// TIA Portal V17 program export: 22 tag tables, 7 data types, 16 data blocks, 26 code blocks (in call order from the OBs), 29 instance data blocks

VAR_GLOBAL   // PLC tag table "Data Costant"
END_VAR
VAR_GLOBAL CONSTANT   // user constants
   MaxCreateNFP : Int := 10;   // Number of max creating NFP²s
   MaxDataReading : Int := 25;   // Number of max data reading
   MaxRoundNumber : Int := 1;   // Number of Rounds
   NumberOfmessages : Int := 6;   // Number of messages from IJCore
   MaxStageStep : Int := 25;   // Number of Max Step Step
   MaxInitStep : Int := 2;   // Number of Max Init Step
   MaxRobot : Int := 3;   // Number of Max Robot
   MaxReader : Int := 5;   // Number of Max Reader
   MaxSolenoid : Int := 48;   // Number of Max Solenoid
   NotUsed : Int := 0;
   MasterNFP : Int := 2;
   SecondaryNFP : Int := 3;
   Component : Int := 4;
   STA : Int := 1;
   PFC : Int := 2;
   TRW : Int := 3;
   TRI : Int := 4;
   TRR : Int := 5;
   CMA : Int := 7;
   TMA : Int := 8;
   CNF : Int := 9;
   TRC : Int := 10;
   TRS : Int := 6;
   TRB : Int := 11;
END_VAR

VAR_GLOBAL   // PLC tag table "Default tag table"
   optoSignal AT %I0.7 : Bool;
   nestScannerBusy AT %I3.0 : Bool;
   nestScannerComplete AT %I4.0 : Bool;
   nestScannerError AT %I5.0 : Bool;
   nestScannerDataSize AT %IW334 : Int;
   upperScannerReading AT %I9.0 : Bool;
   upperScannerReadingComplete AT %I10.0 : Bool;
   upperScannerError AT %I11.0 : Bool;
   upperScannerDataSize AT %IW470 : Int;
   angleScannerDataSize AT %IW385 : Int;
   angleScannerBusy AT %I39.0 : Bool;
   angleScannerReadingComplete AT %I40.0 : Bool;
   angleScannerError AT %I41.0 : Bool;
   amgeScannerDataSize AT %IW606 : Int;
   Tag_1 AT %I46.3 : Bool;
   Tag_2 AT %I46.4 : Bool;
   washerPresence AT %I1.0 : Bool;
   toolingID2 AT %I1.6 : Bool;
   finalTorqueAngle AT %IW17 : Word;
   OutputPin2 AT %QB147 : Byte;
   byte0 AT %QB156 : Byte;
   runlight AT %Q159.2 : Bool;
   byte6 AT %QB162 : Byte;
   byte2 AT %QB158 : Byte;
   byte7 AT %QB163 : Byte;
   segmentLight AT %Q159.0 : Bool;
   byte1 AT %QB157 : Byte;
   byte4 AT %QB160 : Byte;
   byte3 AT %QB159 : Byte;
   byte5 AT %QB161 : Byte;
   optoGreen AT %Q1.2 : Bool;
   optoRed AT %Q1.3 : Bool;
   optoYellow AT %Q1.4 : Bool;
   qYellowTurretBlinking AT %Q2.1 : Bool;
   nestScannerRequest AT %Q3.0 : Bool;
   clearUpperScannerReadComplete AT %Q9.0 : Bool;
   upperScannerRequest AT %Q8.0 : Bool;
   angleScannerRequest AT %Q13.0 : Bool;
   clearAngleScannerComplete AT %Q14.0 : Bool;
   clearTorque AT %Q17.5 : Bool;
   System_Byte AT %MB0 : Byte;
   DiagStatusUpdate AT %M0.1 : Bool;
   "CONFIG INICIAL" AT %M89.5 : Bool;
   "CONFIG CILINDROS ON" AT %M89.7 : Bool;
END_VAR
VAR_GLOBAL CONSTANT   // user constants
   "MODELO MOTOR 1" : String := '592';
   "MODELO MOTOR 2" : String := '202';
   "MODELO MOTOR 3" : String := '277';
   "MODELO MOTOR 4" : String := '984';
   "MODELO TRACK L 1" : String := '610';
   "MODELO TRACK L 2" : String := '618';
   "MODELO TRACK L 3" : String := '333';
   "MODELO TRACK L 4" : String := '444';
   "MODELO TRACK L 5" : String := '555';
   "MODELO TRACK L 6" : String := '666';
   "MODELO TRACK L 7" : String := '777';
   "MODELO TRACK L 8" : String := '888';
   "MODELO TRACK R 1" : String := '612';
   "MODELO TRACK R 2" : String := '623';
   "MODELO TRACK R 3" : String := '993';
   "MODELO TRACK R 4" : String := '994';
   "MODELO TRACK R 5" : String := '995';
   "MODELO TRACK R 6" : String := '996';
   "MODELO TRACK R 7" : String := '997';
   "MODELO TRACK R 8" : String := '998';
END_VAR

VAR_GLOBAL   // PLC tag table "EKSMemory"
   eksUserLevel AT %MB2101 : SInt;
   ActualAuthorizationLevel AT %MB2100 : SInt;
   electronicKeyPresent AT %MB2102 : SInt;
END_VAR

VAR_GLOBAL   // PLC tag table "alarmMemory"
   alarm0 AT %MW100 : Int;   // alarm number
   alarm1 AT %MW102 : Int;   // alarm number
   alarm2 AT %MW104 : Int;
   retIolink AT %MW108 : Int;
   retManifold AT %MW112 : Int;
   retEuchner AT %MW106 : Int;
   retIolink2 AT %MW110 : Int;
   removeScannerError AT %MW6 : Word;
   Green AT %M2.0 : Bool;
   yellow AT %M2.1 : Bool;
   red AT %M2.2 : Bool;
   qRedTurretSolid AT %M3.6 : Bool;
   kkkk AT %M8.1 : Bool;
   hmifinalTorqueAngle AT %MW10 : Word;
END_VAR

VAR_GLOBAL   // PLC tag table "clockMemory"
   Clock_Byte AT %MB1 : Byte;
   Clocks_100ms_FP AT %M1.0 : Bool;
   Clocks_200ms_FP AT %M1.1 : Bool;
   Clocks_400ms_FP AT %M1.2 : Bool;
   Clocks_500ms_FP AT %M1.3 : Bool;
   Clocks_800ms_FP AT %M1.4 : Bool;
   Clocks_1s_FP AT %M1.5 : Bool;
   Clocks_1S600ms_FP AT %M1.6 : Bool;
   Clocks_2s_FP AT %M1.7 : Bool;
END_VAR

VAR_GLOBAL   // PLC tag table "codeReaderMemory"
   reqScannerConfig AT %M2250.2 : Bool;
   bufferReset AT %M2250.0 : Bool;
   labelReadingError AT %M186.3 : Bool;
   labelNok AT %M187.0 : Bool;
   nestLabelReadingError AT %M224.0 : Bool;
   idleTime AT %M2250.1 : Bool;
   seatLabelIdentified AT %M2250.3 : Bool;
   motorLabelIdentified AT %M2250.4 : Bool;
   xLabelIdentified AT %M2250.5 : Bool;
   hmiNestScannerReq AT %M2.3 : Bool;
   scannerOnConfig AT %M2.6 : Bool;
   scanningNest AT %M2.7 : Bool;
   nestCodeRead AT %M3.3 : Bool;
   upperScannerCodeRead AT %M3.4 : Bool;
   angleScannerCodeRead AT %M3.7 : Bool;
   scanningAngle AT %M4.2 : Bool;
   scanningUpper AT %M4.6 : Bool;
   label1Upper AT %M8.2 : Bool;
   label2Upper AT %M8.3 : Bool;
END_VAR

VAR_GLOBAL   // PLC tag table "hmiMemory"
   currentModel AT %MW3000 : Int;
   hmiButtonVisualization AT %M3050.6 : Bool;
   previousModel AT %MW3008 : Int;
   currentStep AT %MW3002 : Int;
   numbersOfStepsToMove AT %MW3006 : UInt;
   stepToDivide AT %MW3012 : UInt;
   stepToInsert AT %MW3014 : UInt;
   hmiScreenNumber AT %MW22 : Int;
   allowedTextChange AT %M3050.0 : Bool;
   progressBarMultiply AT %MW3010 : Int;
   lastCycleInputs AT %MD3034 : DInt;
   energySavingElapsedTime AT %MD3030 : Time;
   f7Button AT %M3050.5 : Bool;
   sequencerCopySequence AT %M66.2 : Bool;
   codeReaderConfigurationVisible AT %M3050.2 : Bool;
   directAlarm AT %M3050.3 : Bool;
   directHome AT %M3050.4 : Bool;
   saveHMI AT %M2.4 : Bool;
   readHMI AT %M2.5 : Bool;
   home AT %M4.7 : Bool;
   ready4Movement AT %M5.5 : Bool;
   popUpVisible AT %M5.6 : Bool;
END_VAR

VAR_GLOBAL   // PLC tag table "modeMemory"
   automaticMode AT %M3.0 : Bool;   // AUTO = 1
   manualMode AT %M3.1 : Bool;
   noMode AT %M3.2 : Bool;
   modelChangePermit AT %M187.1 : Bool;
END_VAR

VAR_GLOBAL   // PLC tag table "permissionMemory"
   MaintenacePermission AT %M4.4 : Bool;
   adminPermission AT %M4.0 : Bool;
   lgPermission AT %M4.5 : Bool;
   gapLeaderUser AT %M4.3 : Bool;
   editingPermission AT %M4.1 : Bool;
   confirmStandby AT %M5.7 : Bool;
   cancelMovement AT %M8.0 : Bool;
END_VAR

VAR_GLOBAL   // PLC tag table "productionMemory"
   shift1Production AT %MW300 : Int;
   shift1 AT %M350.0 : Bool;
   shift2Production AT %MW302 : Int;
   shift2 AT %M350.1 : Bool;
   shift3Production AT %MW304 : Int;
   shift3 AT %M350.2 : Bool;
   timeShift1 AT %M350.3 : Bool;
   timeShift2 AT %M350.4 : Bool;
   timeShift3 AT %M350.5 : Bool;
END_VAR

VAR_GLOBAL   // PLC tag table "programMemory"
   cycleTimeReset AT %M250.1 : Bool;
   clearData AT %M250.0 : Bool;
   productInNest AT %M250.2 : Bool;
   programAutoModeSelection AT %M250.3 : Bool;
END_VAR

VAR_GLOBAL   // PLC tag table "pulses"
   startTighteningPulse1 AT %Q124.0 : Bool;
   hmiPulseInt AT %MD2000 : DInt;
   hmiCycleCounterRestartPulse AT %M2004.4 : Bool;
   model01SelectedPulse AT %M2004.6 : Bool;
   model02SelectedPulse AT %M2004.7 : Bool;
   model03SelectedPulse AT %M2005.0 : Bool;
   model04SelectedPulse AT %M2005.1 : Bool;
   model05SelectedPulse AT %M2005.2 : Bool;
   model06SelectedPulse AT %M2005.3 : Bool;
   model07SelectedPulse AT %M2005.4 : Bool;
   model08SelectedPulse AT %M2005.5 : Bool;
   model09SelectedPulse AT %M2005.6 : Bool;
   model10SelectedPulse AT %M2005.7 : Bool;
   model11SelectedPulse AT %M2006.0 : Bool;
   model12SelectedPulse AT %M2006.1 : Bool;
   mode13SelectedPulse AT %M2006.2 : Bool;
   mode14SelectedPulse AT %M2006.3 : Bool;
   mode15SelectedPulse AT %M2006.4 : Bool;
   alarmPresPulse AT %M2004.3 : Bool;
   "1stShiftChangePulse" AT %M2004.0 : Bool;
   "2ndShiftChangePulse" AT %M2004.1 : Bool;
   "3rdShiftChangePulse" AT %M2004.2 : Bool;
   stepChangeTimerResetInputPulse AT %M2009.4 : Bool;
   stepChangeTimerResetOutputPulse AT %M2009.5 : Bool;
   stationTurnedOffInSequencePulse AT %M2009.3 : Bool;
   model32SelectedPulse AT %M2008.5 : Bool;
   model31SelectedPulse AT %M2008.4 : Bool;
   model30SelectedPulse AT %M2008.3 : Bool;
   model29SelectedPulse AT %M2008.2 : Bool;
   model27SelectedPulse AT %M2008.0 : Bool;
   model28SelectedPulse AT %M2008.1 : Bool;
   model26SelectedPulse AT %M2007.7 : Bool;
   model25SelectedPulse AT %M2007.6 : Bool;
   model24SelectedPulse AT %M2007.5 : Bool;
   model23SelectedPulse AT %M2007.4 : Bool;
   model22SelectedPulse AT %M2007.3 : Bool;
   model21SelectedPulse AT %M2007.2 : Bool;
   model20SelectedPulse AT %M2007.1 : Bool;
   model19SelectedPulse AT %M2007.0 : Bool;
   model18SelectedPulse AT %M2006.7 : Bool;
   model17SelectedPulse AT %M2006.6 : Bool;
   model16SelectedPulse AT %M2006.5 : Bool;
   scanner3DataLogPulse AT %M2009.2 : Bool;
   scanner2DataLogPulse AT %M2009.1 : Bool;
   scanner1DataLogPulse AT %M2009.0 : Bool;
   rightTrackScannerPulse AT %M2008.7 : Bool;
   leftTrackScannerPulse AT %M2004.5 : Bool;
   motorScannerPulse AT %M2008.6 : Bool;
   clearDataPulse AT %M2010.0 : Bool;
   hmiCylinderPulse AT %M5.4 : Bool;
END_VAR

VAR_GLOBAL   // PLC tag table "sequenceMemory"
   aa AT %MW24 : Int;
   a_correctas AT %MW32 : Int;
   a_estados AT %MW34 : Int;
   verificacion_estados_A AT %MW44 : Int;
   verificacion_estados_B AT %MW26 : Int;
   b_estados AT %MW36 : Int;
   numberOfCorrectOutputStates AT %MW38 : Int;
   bb AT %MW40 : Int;
   previousStep AT %MW1112 : Int;
   sequenceRestart AT %M89.1 : Bool;
   stationTurnedOffInSequence AT %M1150.1 : Bool;
END_VAR

VAR_GLOBAL   // PLC tag table "systemMemory"
   firstScan AT %M0.0 : Bool;
   LOG0 AT %M0.3 : Bool;
   LOG1 AT %M0.2 : Bool;
END_VAR

VAR_GLOBAL   // PLC tag table "EKSFieldbusInputs"
   iEKSLevel AT %IB201 : Byte;
   iEKSChipInside AT %I200.1 : Bool;
   iEKSEmpolyeeNumber AT %ID221 : DWord;
   iEKSKeyID1 AT %ID320 : DWord;
   iEKSKeyID2 AT %ID324 : DWord;
   iEKSEmployeeNumber AT %I200.6 : Bool;
   usserIsLogged AT %M2150.0 : Bool;
END_VAR

VAR_GLOBAL   // PLC tag table "powerFocus6000"
   counterClockwiseDirection AT %I182.5 : Bool;
   clockwiseDirection AT %I182.6 : Bool;
   torqueOk AT %I19.6 : Bool;
   torqueDone AT %I20.0 : Bool;
   torqueNok AT %I19.7 : Bool;
   finalTorqueInt1 AT %IW13 : Word;
   finalTorqueDecimal1 AT %IW15 : Word;
   deactivateTool AT %Q17.7 : Bool;
   activateTorqueTool AT %Q17.0 : Bool;
   clearNestScanerRead AT %Q4.0 : Bool;
   torqueInputSelect AT %QB18 : Byte;
   thighteningStart AT %Q17.3 : Bool;
   correctTorque AT %M3.5 : Bool;
   p6000Test1 AT %M152.1 : Bool;
   p6000Test2 AT %M152.2 : Bool;
   p6000Test3 AT %M152.3 : Bool;
   p6000Test1Enabled AT %M152.4 : Bool;
   p6000Test2Enabled AT %M152.5 : Bool;
   p6000Test3Enabled AT %M152.6 : Bool;
   counterClockwiseDirectionWarning AT %M23.0 : Bool;
   clockwiseDirectionWarning AT %M23.1 : Bool;
   hmiFinalTorqueDecimal AT %MW214 : Word;
   hmiFinalTorqueInt AT %MW212 : Word;
END_VAR

VAR_GLOBAL   // PLC tag table "safetyControllerFieldbusInputs"
   isecurityEnabled AT %I46.0 : Bool;
   iEmergencyStop AT %I46.1 : Bool;
   emergencyStopMonitor AT %I46.2 : Bool;
END_VAR

VAR_GLOBAL   // PLC tag table "digitalFieldbusInputs"
   iRightManualRodInsExt AT %I156.5 : Bool;
   iLeftToolingLockExt AT %I1.3 : Bool;
   iRightToolingExt AT %I156.7 : Bool;
   iTorqueToolingExt AT %I156.6 : Bool;
   iRigthManualRodInsRet AT %I157.5 : Bool;
   iLeftToolingLockRet AT %I1.4 : Bool;
   iRightToolingRet AT %I157.7 : Bool;
   iTorqueToolingRet AT %I157.6 : Bool;
   iStrapDetection AT %I45.3 : Bool;
   iLeftBracketDetection AT %I45.2 : Bool;
   iPresLeftManFrame AT %I157.1 : Bool;
   iRightBracketDetection AT %I45.0 : Bool;
   iManualExtOk AT %I158.3 : Bool;
   iProductInsertedLh AT %I45.1 : Bool;
   iLeftHomePos AT %I159.6 : Bool;
   iLeftWorkPos AT %I158.6 : Bool;
   iLeftToolingPos3 AT %I158.7 : Bool;
   iManualExtNok AT %I159.3 : Bool;
   iPresRightPwrFrame AT %I156.3 : Bool;
   iManualBumper AT %I158.5 : Bool;
   iLeftSpringColor AT %I158.2 : Bool;
   iRightSpringColor AT %I158.4 : Bool;
   iLeftManualRodInsRet AT %I157.4 : Bool;
   iInsertionCylindersRet AT %I1.2 : Bool;
   iInsertionCylindersExt AT %I1.1 : Bool;
   iLeftManToolingExtNok AT %I159.7 : Bool;
   iProductInsertedRh AT %I45.6 : Bool;
   iTorqueToolingHome AT %I45.5 : Bool;
   iRightToolinPos1 AT %I156.4 : Bool;
   iRightToolinPos3 AT %I156.2 : Bool;
   iRightToolinPos2 AT %I157.2 : Bool;
   iManualZExtOk AT %I156.0 : Bool;
   iManualZExtNok AT %I157.0 : Bool;
   iRightManToolingRet AT %I158.1 : Bool;
   iTorqueTrigger AT %I160.0 : Bool;
   toolingID1 AT %I1.5 : Bool;
   manualProductPres AT %Q10.0 : Bool;
   powerProductPres AT %Q10.1 : Bool;
END_VAR

VAR_GLOBAL   // PLC tag table "digitalPLCInputs"
   iAirPreassureSensor AT %I0.1 : Bool;
   iPresRightManFrame AT %I156.1 : Bool;
   iRestartButton AT %I0.0 : Bool;
END_VAR

VAR_GLOBAL   // PLC tag table "digitalFieldbusOutputs"
   qcylinder1DirectionA AT %Q149.0 : Bool;
   qcylinder1DirectionB AT %Q151.0 : Bool;
   qcylinder2DirectionA AT %Q149.1 : Bool;
   qcylinder2DirectionB AT %Q151.1 : Bool;
   qcylinder7DirectionA AT %Q701.2 : Bool;
   qcylinder7DirectionB AT %Q701.3 : Bool;
   qcylinder4DirectionA AT %Q149.3 : Bool;
   qcylinder4DirectionB AT %Q151.3 : Bool;
   qcylinder5DirectionA AT %Q149.4 : Bool;
   qcylinder5DirectionB AT %Q151.4 : Bool;
   qcylinder6DirectionA AT %Q149.5 : Bool;
   qcylinder6DirectionB AT %Q151.5 : Bool;
   qcylinder3DirectionA AT %Q149.2 : Bool;
   qcylinder3DirectionB AT %Q151.2 : Bool;
   qcylinder8DirectionA AT %Q701.4 : Bool;
   qcylinder8DirectionB AT %Q701.5 : Bool;
   qcylinder9DirectionA AT %Q701.6 : Bool;
   qcylinder9DirectionB AT %Q701.7 : Bool;
   qcylinder10DirectionA AT %Q702.0 : Bool;
   qcylinder10DirectionB AT %Q702.1 : Bool;
   qActivateCutOffValve AT %Q147.7 : Bool;
END_VAR

VAR_GLOBAL   // PLC tag table "digitalPLCOutputs"
   qAirInletValve1 AT %Q0.0 : Bool;
   qLampActivation AT %Q1.0 : Bool;
   qFanActivation AT %Q1.1 : Bool;
   qControlIN AT %Q1.7 : Bool;
   qAirInletValve2 AT %Q0.1 : Bool;
   qRedTurretBlinking AT %M5.0 : Bool;
   qYellowTurretSolid AT %M5.1 : Bool;
   qGreenTurret AT %M5.2 : Bool;
   qBlueTurret AT %M5.3 : Bool;
END_VAR

VAR_GLOBAL   // PLC tag table "EKSFieldbusOutputs"
   qEKSStartAddress AT %QB201 : Byte;
   qEKSDataLength AT %QB202 : Byte;
   qEKSData1 AT %QB204 : Byte;
   qEKSData2 AT %QB205 : Byte;
   qEKsWriteCMD AT %Q200.0 : Bool;
END_VAR

TYPE "UDT_Readings"
// stored: IsFailsafeCompliant false
   STRUCT
      Enable : Bool;   // Reading active
      ReaderNumber : USInt;   // Fix (1 to 5) or Manual (10)
      "Name" : String[30];   // Name of Label to read
      LabelType : USInt;   // Master NFP, 2nd NFP, Component Label, batch label
      ReferenceToFound : String[30];   // Reference to be found
      ReferenceStartPosition : USInt;   // Position of reference to be found
      ReferenceLenght : USInt;   // Reference Lenght
      MasterReadingNumber : USInt;   // Reading number of master NFP
      LinkedMasterNumber : USInt;   // Linked number to master NFP
      Message : Array[1.."NumberOfmessages"] of "UDT_IJCoreMessage";   // IJCore Message
   END_STRUCT;
END_TYPE

TYPE "UDT_ScrewData"
// stored: IsFailsafeCompliant false
   STRUCT
      Torque : Struct   // Torque Data
         BeforePoint : Word;   // Torque before point
         AfterPoint : Word;   // Torque after point
      END_STRUCT;
      Angle : Word;   // angle
   END_STRUCT;
END_TYPE

TYPE "udtButtons"
// stored: IsFailsafeCompliant false
   STRUCT
      bReq : Bool;
      bP : Bool;
      bTGG : Bool;
      bCmd : Bool;
      bAkn : Bool;
      b1 : Bool;
      b2 : Bool;
      b3 : Bool;
   END_STRUCT;
END_TYPE

TYPE "udt_EKS_KEY"
// stored: IsFailsafeCompliant false
   STRUCT
      ID1 : DWord;   // Key unique ID [bytes 1-4]
      ID2 : DWord;   // Key unique ID [bytes 5-8]
      EMPLOYEE_ID : DWord;   // Employee ID number [hex format]
      LEVEL : Int;   // Key level stored inside key
      COMMENTS : WString[10];   // Comments of the key
      _res_1 : Int;
   END_STRUCT;
END_TYPE

TYPE "udt_referenceMainInfo"
// stored: IsFailsafeCompliant false
   STRUCT
      id : Int;
      description : String[20];
      partNumber : String[8];
      rev : String[2];
      customerNumber : String[8];
      vpps : String[14];
      locationCode : String[1];
      dataIdentifier : String[3];
      duns : String[9];
   END_STRUCT;
END_TYPE

TYPE "CONFIG_MSG_IJC"
// stored: IsFailsafeCompliant false
   STRUCT
      "TYPE" : String[3];
      KANBAN : String[30];
      COMPONENT : String[62];
      START : Bool;
      PROCESS_STATUS : SInt;
   END_STRUCT;
END_TYPE

TYPE "UDT_IJCoreMessage"
// stored: IsFailsafeCompliant false
   STRUCT
      MessageType : USInt;
      MessageFlagNumber : UInt;
      SendMsg : Bool;
      Done : Bool;
      Answer : Int;
      State : USInt;
   END_STRUCT;
END_TYPE

DATA_BLOCK "DB_MAIN_IJCORE"   // DB1000
{ S7_Optimized_Access := 'FALSE' }
VERSION : 0.1
// stored: AutoNumber false, DBAccessibleFromOPCUA true, DBAccessibleFromWebserver true, IsOnlyStoredInLoadMemory false, IsWriteProtectedInAS false
   VAR
      Enable : Bool := true;   // Enable traceability
      Mode : USInt := 1;   // 1. Full traceability, 2. Downgrade Mode
      Errors : Word;   // Error code
      hmiInd : USInt;   // Global Indicator Status
      CreatedNFP : Array[1.."MaxCreateNFP"] of String[30];   // Created NFP
      STAT : Struct
         STA_OK : Bool;
         PFC_OK : Bool;
         TRC_OK : Bool;
         CNF_OK : Bool;
         TRR_OK : Bool;
         ProcessResults : USInt;   // 1: Part OK, 2: PartNOK
      END_STRUCT;
      CMD : Struct
         STA : Bool;
         PFC : Bool;
         TRC : Bool;
         CNF : Bool;
         TRR : Bool;
      END_STRUCT;
   END_VAR
BEGIN
END_DATA_BLOCK

DATA_BLOCK "DB_REC_IJCORE"   // DB1006
{ S7_Optimized_Access := 'FALSE' }
VERSION : 0.1
// stored: AutoNumber false, DBAccessibleFromOPCUA true, DBAccessibleFromWebserver true, IsOnlyStoredInLoadMemory false, IsWriteProtectedInAS false
   VAR
      SW_Message : Array[1..300] of Word;
      Message : Array[1..50] of Struct
         Answer : Int;
         Content : Array[1..30] of Byte;
      END_STRUCT;
   END_VAR
BEGIN
END_DATA_BLOCK

DATA_BLOCK "DB_SEND_IJCORE"   // DB1005
{ S7_Optimized_Access := 'FALSE' }
VERSION : 0.1
// stored: AutoNumber false, DBAccessibleFromOPCUA true, DBAccessibleFromWebserver true, IsOnlyStoredInLoadMemory false, IsWriteProtectedInAS false
   VAR
      Awake_DW : Word;
      Awake_SW : Int;
      SW_Message : Array[1..300] of Word;
      Message : Array[1..50] of Struct
         Content : Array[1..80] of Byte;
      END_STRUCT;
   END_VAR
BEGIN
END_DATA_BLOCK

DATA_BLOCK "DB_EKS"   // DB305
{ S7_Optimized_Access := 'FALSE' }
VERSION : 0.1
// stored: AutoNumber false, DBAccessibleFromOPCUA true, DBAccessibleFromWebserver true, IsOnlyStoredInLoadMemory false, IsWriteProtectedInAS false
   VAR RETAIN
      STAT : Struct
         OPERATOR : Bool := TRUE;
         GAP_LEADER : Bool := TRUE;
         MAINTENANCE : Bool := TRUE;
         ADMINISTRATOR : Bool := TRUE;
         _4 : Bool := FALSE;
         _5 : Bool := FALSE;
         _6 : Bool := FALSE;
         _7 : Bool := FALSE;
         ADD_MODE_ENABLED : Bool := TRUE;
         ADD_MODE : Bool := FALSE;
         RESET : Bool := FALSE;
         NB_MAX_ACHIEVED : Bool := FALSE;
         FP_STORE_KEY_IN : Bool := FALSE;
         _15 : Bool := FALSE;
         _16 : Bool := FALSE;
         _17 : Bool := FALSE;
      END_STRUCT;
      HMI : Struct
         OPERATOR_KEY : Bool := FALSE;
         ADD_MODE : Bool := FALSE;
         END_ADD_MODE : Bool := FALSE;
         WRITE_NEW_KEY_LEVEL : Bool := FALSE;
         WRITE_NEW_KEY_ID : Bool := FALSE;
         UPDATE_NB_ADMIN : Bool := FALSE;
         _6 : Bool := FALSE;
         _7 : Bool := FALSE;
         _10 : Bool := FALSE;
         _11 : Bool := FALSE;
         _12 : Bool := FALSE;
         _13 : Bool := FALSE;
         _14 : Bool := FALSE;
         _15 : Bool := FALSE;
         _16 : Bool := FALSE;
         _17 : Bool := FALSE;
      END_STRUCT;
      TIM : Struct
         RESET_SET : Int := 9999;
         RESET_STAT : Int := 2960;
      END_STRUCT;
      PAGE_INDEX : Int := 1;   // Index of the page of HMI
      SAVE_LINE : Int := 0;   // Line to save key
      REMOVE_LINE : Int := 0;   // Line to remove key
      ACTUAL_LEVEL : Int := 5;   // Actual level of key
      NB_ADMIN : Int := 27414;   // Number of admin counted
      T_CYCLE : Int := 0;   // Index for function Cycle (look for key)
      NB_MAX_ADMIN : Int := 5;   // Number of administrator max
      Number_page_saved : Word := 16#0001;
      _res : Array[22..47] of Byte;   // Reserve
      INSERTED_KEY { S7_SetPoint := 'True'} : "udt_EKS_KEY";   // Information of Key Inserted
      HMI_PAGE { S7_SetPoint := 'True'} : Array[1..10] of "udt_EKS_KEY";   // Information displayed on HMI
      _res_1 : Array[270..299] of Byte;   // Reserve
      KEYS { S7_SetPoint := 'True'} : Array[1..130] of "udt_EKS_KEY";
      DELETE_KEY : "udt_EKS_KEY";
   END_VAR
BEGIN
   _res[22..47] := 16#00;
   INSERTED_KEY.ID1 := 16#383E_0010;
   INSERTED_KEY.ID2 := 16#3200_0000;
   INSERTED_KEY.EMPLOYEE_ID := 16#0000_0000;
   INSERTED_KEY.LEVEL := 5;
   INSERTED_KEY.COMMENTS := WSTRING#'LIMON';
   INSERTED_KEY._res_1 := 0;
   HMI_PAGE[1].ID1 := 16#2B2F_0010;
   HMI_PAGE[2].ID1 := 16#28A5_0010;
   HMI_PAGE[3].ID1 := 16#0000_0000;
   HMI_PAGE[4].ID1 := 16#71A6_0010;
   HMI_PAGE[5].ID1 := 16#8037_0010;
   HMI_PAGE[6].ID1 := 16#383E_0010;
   HMI_PAGE[7].ID1 := 16#5A1E_0010;
   HMI_PAGE[8].ID1 := 16#D65A_0010;
   HMI_PAGE[9..10].ID1 := 16#0000_0000;
   HMI_PAGE[1..2].ID2 := 16#3200_0000;
   HMI_PAGE[3].ID2 := 16#0000_0000;
   HMI_PAGE[4..8].ID2 := 16#3200_0000;
   HMI_PAGE[9..10].ID2 := 16#0000_0000;
   HMI_PAGE[1..7].EMPLOYEE_ID := 16#0000_0000;
   HMI_PAGE[8].EMPLOYEE_ID := 16#0000_0001;
   HMI_PAGE[9..10].EMPLOYEE_ID := 16#0000_0000;
   HMI_PAGE[1].LEVEL := 5;
   HMI_PAGE[2].LEVEL := 3;
   HMI_PAGE[3].LEVEL := 0;
   HMI_PAGE[4].LEVEL := 2;
   HMI_PAGE[5].LEVEL := 3;
   HMI_PAGE[6].LEVEL := 5;
   HMI_PAGE[7].LEVEL := 3;
   HMI_PAGE[8].LEVEL := 2;
   HMI_PAGE[9..10].LEVEL := 0;
   HMI_PAGE[1].COMMENTS := WSTRING#'CLAUDIO';
   HMI_PAGE[2].COMMENTS := WSTRING#'CLAUDIO-M';
   HMI_PAGE[3].COMMENTS := WSTRING#'';
   HMI_PAGE[4].COMMENTS := WSTRING#'GAP-1';
   HMI_PAGE[5].COMMENTS := WSTRING#'MANT-1';
   HMI_PAGE[6].COMMENTS := WSTRING#'LIMON';
   HMI_PAGE[7].COMMENTS := WSTRING#'MANT';
   HMI_PAGE[8].COMMENTS := WSTRING#'GAP';
   HMI_PAGE[9..10].COMMENTS := WSTRING#'';
   HMI_PAGE[1..10]._res_1 := 0;
   _res_1[270..299] := 16#00;
   KEYS[1].ID1 := 16#2B2F_0010;
   KEYS[2].ID1 := 16#28A5_0010;
   KEYS[3].ID1 := 16#0000_0000;
   KEYS[4].ID1 := 16#71A6_0010;
   KEYS[5].ID1 := 16#8037_0010;
   KEYS[6].ID1 := 16#383E_0010;
   KEYS[7].ID1 := 16#5A1E_0010;
   KEYS[8].ID1 := 16#D65A_0010;
   KEYS[9..109].ID1 := 16#0000_0000;
   KEYS[110].ID1 := 16#DB52_0010;
   KEYS[111..130].ID1 := 16#0000_0000;
   KEYS[1..2].ID2 := 16#3200_0000;
   KEYS[3].ID2 := 16#0000_0000;
   KEYS[4..8].ID2 := 16#3200_0000;
   KEYS[9..109].ID2 := 16#0000_0000;
   KEYS[110].ID2 := 16#3200_0000;
   KEYS[111..130].ID2 := 16#0000_0000;
   KEYS[1..7].EMPLOYEE_ID := 16#0000_0000;
   KEYS[8].EMPLOYEE_ID := 16#0000_0001;
   KEYS[9..130].EMPLOYEE_ID := 16#0000_0000;
   KEYS[1].LEVEL := 5;
   KEYS[2].LEVEL := 3;
   KEYS[3].LEVEL := 0;
   KEYS[4].LEVEL := 2;
   KEYS[5].LEVEL := 3;
   KEYS[6].LEVEL := 5;
   KEYS[7].LEVEL := 3;
   KEYS[8].LEVEL := 2;
   KEYS[9..109].LEVEL := 0;
   KEYS[110].LEVEL := 5;
   KEYS[111..130].LEVEL := 0;
   KEYS[1].COMMENTS := WSTRING#'CLAUDIO';
   KEYS[2].COMMENTS := WSTRING#'CLAUDIO-M';
   KEYS[3].COMMENTS := WSTRING#'';
   KEYS[4].COMMENTS := WSTRING#'GAP-1';
   KEYS[5].COMMENTS := WSTRING#'MANT-1';
   KEYS[6].COMMENTS := WSTRING#'LIMON';
   KEYS[7].COMMENTS := WSTRING#'MANT';
   KEYS[8].COMMENTS := WSTRING#'GAP';
   KEYS[9..109].COMMENTS := WSTRING#'';
   KEYS[110].COMMENTS := WSTRING#'Robins';
   KEYS[111..130].COMMENTS := WSTRING#'';
   KEYS[1..130]._res_1 := 0;
   DELETE_KEY.ID1 := 16#0000_0000;
   DELETE_KEY.ID2 := 16#0000_0000;
   DELETE_KEY.EMPLOYEE_ID := 16#0000_0000;
   DELETE_KEY.LEVEL := 0;
   DELETE_KEY.COMMENTS := WSTRING#'';
   DELETE_KEY._res_1 := 0;
END_DATA_BLOCK

DATA_BLOCK "LABELS"   // DB6
{ S7_Optimized_Access := 'TRUE' }
VERSION : 0.1
// stored: AutoNumber false, DBAccessibleFromOPCUA true, DBAccessibleFromWebserver true, IsOnlyStoredInLoadMemory false, IsRetainMemResEnabled false, IsWriteProtectedInAS false, MemoryReserve 100
   VAR
      "Previous code" : String := '[) 06 Y40.02.07.01.L P8127005 12V812785841 T9T22202A2B4C1004';
      "Result comp 3" : Int := 0;
      "Result comp 2" : Int := 0;
      "Result comp 1" : Int := 0;
      "Label comp 3" : String := '';
      "Label comp 2" : String := '';
      "Label comp 1" : String := '15';
   END_VAR
   VAR RETAIN
      "Label 1" : Array[0..16] of String[5];   // Label 1
      "Label 2" { ExternalVisible := 'False'} : Array[0..16] of String[5];
      "Label 3" : Array[0..16] of String[5];
      "Label 4" : Array[0..16] of String[5];
      "Label 5" : Array[0..16] of String[5];
      "Label Pos 1" : Array[0..16] of Int;   // label position 1
      "Label Pos 2" : Array[0..16] of Int;
      "Label Pos 3" : Array[0..16] of Int;
      "Label Pos 4" : Array[0..16] of Int;
      "Label Pos 5" : Array[0..16] of Int;   // label position 2
      "Label int" : Array[0..16] of Int;
      Text : Array[0..16] of String[10];   // label text hmi
   END_VAR
   VAR
      Done : Bool := FALSE;
      "Port error" : Bool := FALSE;
      "Port status" : Word := 16#7000;
      "Reset status" : Word := 16#7000;
   END_VAR
   VAR RETAIN
      "Reset done" : Bool := FALSE;
      scanner1 : Bool := TRUE;
      scanner2 : Bool := TRUE;
      scanner3 : Bool := TRUE;
      scanner4 : Bool := FALSE;
      scanner5 : Bool := FALSE;
      scanner6 : Bool := FALSE;
   END_VAR
   VAR
      scannerOn : Bool := TRUE;
      "scann code" : Array[0..1] of String[30];
      "Recive code 2" : String[80] := '';
      labelPrint : String[20] := 'CR24032821X05357';
      NFP : String[35] := '';
      "Recive code" : String[80] := '';
      NDR : Bool := FALSE;
      Error : Bool := FALSE;
      Status : Word := 16#7002;
      Length : UInt := 0;
      labelBlock : Array[0..6] of Bool;
      "Reading scann 1" : String[180] := '';
      "Reading scann 2" : String[180] := 'V008345Y4259698XR011464240801';
      "Extract 5" : Array[0..16] of String[10];
      "Extract 4" : Array[0..16] of String[10];
      "Extract 3" : Array[0..16] of String[10];
      "Extract 2" : Array[0..16] of String[10];
      "Extract 1" : Array[0..16] of String[10];
      "Scanner reading" : Array[0..254] of Char;
      "Previous code scann" : String[40] := '';
      scannerOK2 : Bool := FALSE;
      scannerOK3 : Bool := FALSE;
      scannerOK4 : Bool := FALSE;
      scannerOK5 : Bool := FALSE;
      ScannerOK1 : Bool := FALSE;
      "Scanner length 5" : Array[0..16] of Int;
      "Scanner length 4" : Array[0..16] of Int;
      "Scanner length 3" : Array[0..16] of Int;
      "Scanner length 2" : Array[0..16] of Int;
      "Scanner length 1" : Array[0..16] of Int;
      nestCodeRead : String[80] := '';
      upperCodeRead : String[80] := '';
      angleCodeRead : String[80] := '';
   END_VAR
BEGIN
   "Label 1"[0] := '695';
   "Label 1"[1] := '698';
   "Label 1"[2] := '695';
   "Label 1"[3] := '721';
   "Label 1"[4] := '8721X';
   "Label 1"[5..6] := '698';
   "Label 1"[7..16] := '';
   "Label 2"[0..3] := '06';
   "Label 2"[4] := '1';
   "Label 2"[5] := '06';
   "Label 2"[6] := 'Y4';
   "Label 2"[7..16] := '';
   "Label 3"[0..3] := '06';
   "Label 3"[4] := '';
   "Label 3"[5] := '06';
   "Label 3"[6..16] := '';
   "Label 4"[0..3] := 'Y4';
   "Label 4"[4] := '5/';
   "Label 4"[5] := 'Y4';
   "Label 4"[6] := '5/';
   "Label 4"[7..16] := '';
   "Label 5"[0..6] := '5/';
   "Label 5"[7..16] := '';
   "Label Pos 1"[0..3] := 13;
   "Label Pos 1"[4] := 12;
   "Label Pos 1"[5..6] := 13;
   "Label Pos 1"[7..16] := 0;
   "Label Pos 2"[0..3] := 4;
   "Label Pos 2"[4] := 1;
   "Label Pos 2"[5] := 4;
   "Label Pos 2"[6] := 1;
   "Label Pos 2"[7..16] := 0;
   "Label Pos 3"[0..3] := 4;
   "Label Pos 3"[4] := 0;
   "Label Pos 3"[5] := 4;
   "Label Pos 3"[6..16] := 0;
   "Label Pos 4"[0..3] := 1;
   "Label Pos 4"[4] := 20;
   "Label Pos 4"[5] := 1;
   "Label Pos 4"[6] := 20;
   "Label Pos 4"[7..16] := 0;
   "Label Pos 5"[0..6] := 20;
   "Label Pos 5"[7..16] := 0;
   "Label int"[0] := 151;
   "Label int"[1..16] := 0;
   Text[0] := '';
   Text[1] := 'NEST';
   Text[2] := 'UPPER1';
   Text[3] := 'ANGLE';
   Text[4] := 'UPPER2';
   Text[5..16] := '';
   "scann code"[0..1] := '';
   labelBlock[0..6] := FALSE;
   "Extract 5"[0..16] := '';
   "Extract 4"[0..16] := '';
   "Extract 3"[0..16] := '';
   "Extract 2"[0..16] := '';
   "Extract 1"[0..16] := '';
   "Scanner reading"[0] := '$L';
   "Scanner reading"[1] := '†';
   "Scanner reading"[2] := '$L';
   "Scanner reading"[3] := '†';
   "Scanner reading"[4] := '$L';
   "Scanner reading"[5] := '†';
   "Scanner reading"[6] := '$00';
   "Scanner reading"[7] := '$1E';
   "Scanner reading"[8] := 'B';
   "Scanner reading"[9..10] := '0';
   "Scanner reading"[11] := '2';
   "Scanner reading"[12] := '3';
   "Scanner reading"[13] := '9';
   "Scanner reading"[14] := '0';
   "Scanner reading"[15] := 'W';
   "Scanner reading"[16] := '4';
   "Scanner reading"[17] := '2';
   "Scanner reading"[18] := '6';
   "Scanner reading"[19] := '8';
   "Scanner reading"[20] := '7';
   "Scanner reading"[21] := '2';
   "Scanner reading"[22] := '1';
   "Scanner reading"[23] := 'X';
   "Scanner reading"[24] := 'R';
   "Scanner reading"[25] := '0';
   "Scanner reading"[26..27] := '1';
   "Scanner reading"[28] := '4';
   "Scanner reading"[29] := '6';
   "Scanner reading"[30] := '4';
   "Scanner reading"[31] := '2';
   "Scanner reading"[32] := '4';
   "Scanner reading"[33] := '0';
   "Scanner reading"[34] := '2';
   "Scanner reading"[35] := '0';
   "Scanner reading"[36] := '1';
   "Scanner reading"[37] := '$R';
   "Scanner reading"[38..135] := '$00';
   "Scanner reading"[136..254] := ' ';
   "Scanner length 5"[0] := 0;
   "Scanner length 5"[1] := 3;
   "Scanner length 5"[2..16] := 0;
   "Scanner length 4"[0] := 0;
   "Scanner length 4"[1] := 3;
   "Scanner length 4"[2..16] := 0;
   "Scanner length 3"[0] := 0;
   "Scanner length 3"[1] := 3;
   "Scanner length 3"[2..16] := 0;
   "Scanner length 2"[0] := 0;
   "Scanner length 2"[1] := 3;
   "Scanner length 2"[2..16] := 0;
   "Scanner length 1"[0] := 5;
   "Scanner length 1"[1] := 3;
   "Scanner length 1"[2..16] := 0;
END_DATA_BLOCK

DATA_BLOCK "Conveyor_DB"   // DB41
{ S7_Optimized_Access := 'FALSE' }
VERSION : 0.1
// stored: AutoNumber true, DBAccessibleFromOPCUA true, DBAccessibleFromWebserver true, IsOnlyStoredInLoadMemory false, IsWriteProtectedInAS false
   VAR
      printLabel : Bool := FALSE;
      description : String := 'BACKREST W33A POWER MEMO L6';
      partNumber : String := '2389161X-01';
      lastScann : String := '038040781M41839';
      okModelBit : Bool := FALSE;
      leftTrackScan : String := 'JI2U07619706';
      rightTrackScan : String := 'FR2I01420707';
      motorScan : String := '038040781M41839';
   END_VAR
BEGIN
END_DATA_BLOCK

DATA_BLOCK "Data_logging"   // DB36
{ S7_Optimized_Access := 'TRUE' }
VERSION : 0.1
// stored: AutoNumber true, DBAccessibleFromOPCUA true, DBAccessibleFromWebserver true, IsOnlyStoredInLoadMemory false, IsRetainMemResEnabled false, IsWriteProtectedInAS false, MemoryReserve 100
   VAR
      scanning : Array[1..3] of String;
      alignment : Real := 0.0;
      pieceOk : Bool := FALSE;
   END_VAR
BEGIN
   scanning[1] := '038040781M41839';
   scanning[2] := 'JI2U07619706';
   scanning[3] := 'FR2I01420707';
END_DATA_BLOCK

DATA_BLOCK "torque"   // DB34
{ S7_Optimized_Access := 'TRUE' }
VERSION : 0.1
// stored: AutoNumber true, DBAccessibleFromOPCUA true, DBAccessibleFromWebserver true, IsOnlyStoredInLoadMemory false, IsRetainMemResEnabled false, IsWriteProtectedInAS false, MemoryReserve 100
   VAR
      ON : Bool := FALSE;
      SENSOR : Int := 0;
      TORQUE : Int := 0;
      TIMER1 { S7_SetPoint := 'True'} : TON_TIME;
      TIMER2 { S7_SetPoint := 'True'} : TON_TIME;
      TIMER3 { S7_SetPoint := 'True'} : TON_TIME;
      TIMER4 { S7_SetPoint := 'True'} : TON_TIME;
      TIMER5 { S7_SetPoint := 'True'} : TON_TIME;
      "1stInt" : Word := 16#0000;
      "2ndInt" : Word := 16#0000;
      "3rdInt" : Word := 16#0000;
      "4thInt" : Word := 16#0000;
      "5thInt" : Word := 16#0000;
      "1stDecimal" : Word := 16#0000;
      "2ndDecimal" : Word := 16#0000;
      "3rdDecimal" : Word := 16#0000;
      "4thDecimal" : Word := 16#0000;
      "5thDecimal" : Word := 16#0000;
      "1stFinalAngle" : Word := 16#0000;
      "2ndFinalAngle" : Word := 16#0000;
      "3rdFinalAngle" : Word := 16#0000;
      "4thFinalAngle" : Word := 16#0000;
      "5thFinalAngle" : Word := 16#0000;
      "ENTERO MANUAL" : Word := 16#0000;
      "DECIMAL MANUAL" : Word := 16#0000;
      "ANGULO FINAL MANUAL" : Word := 16#0000;
      TORNILLO : Int := 0;
      "1Ok" : Bool := FALSE;
      "2Ok" : Bool := FALSE;
      "3Ok" : Bool := FALSE;
      "4Ok" : Bool := FALSE;
      "1_OK_2" : Bool := FALSE;
      "2_OK_2" : Bool := FALSE;
      "3_OK_2" : Bool := FALSE;
      "4_OK_2" : Bool := FALSE;
      "5_OK_2" : Bool := FALSE;
      "5_OK" : Bool := FALSE;
      "ACTIVAR MANUAL" : Bool := FALSE;
      "CONFIG1 MANUAL" : Bool := FALSE;
      "CONFIG2 MANUAL" : Bool := FALSE;
      "CONFIG3 MANUAL" : Bool := FALSE;
      "CONFIG4 MANUAL" : Bool := FALSE;
      "CONFIG5 MANUAL" : Bool := FALSE;
      "REINICIAR PFJOB" : Bool := FALSE;
      PRESET1 : Int := 0;
      PRESET2 : Int := 0;
      PRESET3 : Int := 0;
      PRESET4 : Int := 0;
      PRESET5 : Int := 0;
      manual2 : Struct
         HABILITAR : Bool := TRUE;
         DESHABILITAR : Bool := FALSE;
         BORRAR : Bool := FALSE;
      END_STRUCT;
      BLOQUEO : Array[0..6] of Bool;
      manual : Struct
         activate : Bool := TRUE;
         deactivate : Bool := FALSE;
         erase : Bool := FALSE;
      END_STRUCT;
   END_VAR
   VAR RETAIN
      "P6000 TORQUE_1" : Array[0..15] of Int;
      p6000Torque : Array[0..15] of Int;
   END_VAR
   VAR
      nok2 : Array[0..1] of Bool;
      nok : Array[0..1] of Bool;
   END_VAR
BEGIN
   TIMER1.PT := T#0MS;
   TIMER1.IN := FALSE;
   TIMER2.PT := T#0MS;
   TIMER2.IN := FALSE;
   TIMER3.PT := T#0MS;
   TIMER3.IN := FALSE;
   TIMER4.PT := T#0MS;
   TIMER4.IN := FALSE;
   TIMER5.PT := T#0MS;
   TIMER5.IN := FALSE;
   BLOQUEO[0..6] := FALSE;
   "P6000 TORQUE_1"[0] := 1;
   "P6000 TORQUE_1"[1] := 2;
   "P6000 TORQUE_1"[2] := 3;
   "P6000 TORQUE_1"[3] := 1;
   "P6000 TORQUE_1"[4] := 2;
   "P6000 TORQUE_1"[5] := 3;
   "P6000 TORQUE_1"[6..15] := 0;
   p6000Torque[0] := 1;
   p6000Torque[1] := 2;
   p6000Torque[2] := 3;
   p6000Torque[3] := 1;
   p6000Torque[4] := 2;
   p6000Torque[5] := 3;
   p6000Torque[6..15] := 0;
   nok2[0..1] := FALSE;
   nok[0..1] := FALSE;
END_DATA_BLOCK

DATA_BLOCK "DB_HMI"   // DB7
{ S7_Optimized_Access := 'TRUE' }
VERSION : 0.1
// stored: AutoNumber true, DBAccessibleFromOPCUA true, DBAccessibleFromWebserver true, IsOnlyStoredInLoadMemory false, IsRetainMemResEnabled false, IsWriteProtectedInAS false, MemoryReserve 100
   VAR
      modeButton : Bool := FALSE;
      mode : Int := 2;
      model : Array[0..32] of Bool;
      recipeStep : Int := 3;
      "a" : DInt := -2_146_096_376;
      "b" : DInt := 4197;
      mascA : DInt := 134_221_952;
      mascB : DInt := 0;
      recipeStepTime : Int := 500;
      recipeStepSubstract : Bool := FALSE;
      recipeStepAdd : Bool := FALSE;
      recipeLastStep : Int := 3;
      updateStep : Bool := FALSE;
      moveToCurrentStep : Bool := FALSE;
      recordA1 : Bool := FALSE;
      readA1 : Bool := FALSE;
      recordA2 : Bool := FALSE;
      readA2 : Bool := FALSE;
      recordB1 : Bool := FALSE;
      readB1 : Bool := FALSE;
      recordB2 : Bool := FALSE;
      readB2 : Bool := FALSE;
      recordAnalog : Bool := FALSE;
      readAnalog : Bool := FALSE;
      recipeStepQuantity : Int := 8;
      eraseStep : Bool := FALSE;
      insertStep : Bool := FALSE;
      copyStep : Bool := FALSE;
      copySequence : Bool := FALSE;
      copySequenceStep : Bool := FALSE;
      baseStep : Int := 7;
      destinationStep : Int := 8;
      baseModel : Int := 3;
      destinationModel : Int := 6;
      baseModelStep : Int := 0;
      modelDestinationStep : Int := 0;
      baseModelStep_1 : Int := 2;
      modelDestinationStep_1 : Int := 3;
      operatorTextIndicator : String := ' ';
      enableStationAir : Bool := FALSE;
      enableAirHmiPermission : Bool := FALSE;
      insertAlarmKey : Bool := FALSE;
      enableStationVisualizationButton : Bool := FALSE;
      enableStationHideAlarmButton : Bool := FALSE;
      alarmAckmowledge : Bool := FALSE;
      home : Bool := FALSE;
      advancePercentage : Real := 0.0;
      administratorAlarmButton : Bool := FALSE;
      activateLamp : Bool := TRUE;
      activateFan : Bool := TRUE;
   END_VAR
   VAR RETAIN
      cicles : Int := 285;
      production1 : Int := 247;
      production2 : Int := 56;
      production3 : Int := 0;
   END_VAR
   VAR
      productionRestart1 : Bool := FALSE;
      productionRestart2 : Bool := FALSE;
      productionRestart3 : Bool := FALSE;
      ciclesRestart : Bool := FALSE;
      manualPrint : Bool := FALSE;
      BLOQUEO : Bool := TRUE;
      manualModeNecessary : Bool := FALSE;
      modelChange : Bool := FALSE;
      alarmManualButton : Bool := FALSE;
      user : String := 'Administrator';
      pass : String := 'PASSWORD';
   END_VAR
BEGIN
   model[0..32] := FALSE;
END_DATA_BLOCK

DATA_BLOCK "sensorDistribution"   // DB129
{ S7_Optimized_Access := 'TRUE' }
VERSION : 0.1
// stored: AutoNumber false, DBAccessibleFromOPCUA true, DBAccessibleFromWebserver true, IsOnlyStoredInLoadMemory false, IsRetainMemResEnabled false, IsWriteProtectedInAS false, MemoryReserve 100
   VAR
      inputsStatus : Array[0..31] of Byte;
      outputsStatus : Array[0..31] of Byte;
   END_VAR
BEGIN
   inputsStatus[0..1] := 16#00;
   inputsStatus[2] := 16#01;
   inputsStatus[3..7] := 16#00;
   inputsStatus[8..9] := 16#01;
   inputsStatus[10] := 16#00;
   inputsStatus[11..13] := 16#01;
   inputsStatus[14..16] := 16#00;
   inputsStatus[17..18] := 16#01;
   inputsStatus[19..23] := 16#00;
   inputsStatus[24] := 16#01;
   inputsStatus[25..30] := 16#00;
   inputsStatus[31] := 16#01;
   outputsStatus[0] := 16#00;
   outputsStatus[1] := 16#01;
   outputsStatus[2] := 16#00;
   outputsStatus[3] := 16#01;
   outputsStatus[4] := 16#00;
   outputsStatus[5] := 16#01;
   outputsStatus[6] := 16#00;
   outputsStatus[7] := 16#01;
   outputsStatus[8..12] := 16#00;
   outputsStatus[13] := 16#01;
   outputsStatus[14..31] := 16#00;
END_DATA_BLOCK

DATA_BLOCK "RETENTIVE"   // DB54
{ S7_Optimized_Access := 'TRUE' }
VERSION : 0.1
// stored: AutoNumber true, DBAccessibleFromOPCUA true, DBAccessibleFromWebserver true, IsOnlyStoredInLoadMemory false, IsRetainMemResEnabled true, IsWriteProtectedInAS false, MemoryReserve 100, RetainMemoryReserve 0
   VAR RETAIN
      stationInSequence : Bool := FALSE;
   END_VAR
BEGIN
END_DATA_BLOCK

DATA_BLOCK "STEP"   // DB4
{ S7_Optimized_Access := 'TRUE' }
VERSION : 0.1
// stored: AutoNumber false, DBAccessibleFromOPCUA true, DBAccessibleFromWebserver true, IsOnlyStoredInLoadMemory false, IsRetainMemResEnabled false, IsWriteProtectedInAS false, MemoryReserve 100
   VAR RETAIN
      "time" : Array[0..32, 0..25] of Int;   // Tiempo de duración de cada paso [modelo, paso]
      number : Array[0..32] of Int;   // Número de pasos por modelo
   END_VAR
   VAR
      stepChangeTimer : DInt := 500;
      stepChangeTimerStart : Bool := FALSE;
      counterDone : Bool := FALSE;
   END_VAR
BEGIN
   "time"[0,0..7] := 500;
   "time"[0,8..25] := 0;
   "time"[1,0..7] := 500;
   "time"[1,8..25] := 0;
   "time"[2,0..7] := 500;
   "time"[2,8..25] := 0;
   "time"[3,0..6] := 500;
   "time"[3,7..25] := 0;
   "time"[4,0..6] := 500;
   "time"[4,7..25] := 0;
   "time"[5,0..6] := 500;
   "time"[5,7..25] := 0;
   "time"[6,0..6] := 500;
   "time"[6,7..25] := 0;
   "time"[7,0] := 0;
   "time"[7,1..2] := 1500;
   "time"[7,3] := 0;
   "time"[7,4..9] := 3000;
   "time"[7,10..25] := 0;
   "time"[8,0] := 0;
   "time"[8,1..2] := 1500;
   "time"[8,3] := 0;
   "time"[8,4..9] := 3000;
   "time"[8,10..25] := 0;
   "time"[9,0..3] := 0;
   "time"[9,4..5] := 500;
   "time"[9,6..25] := 0;
   "time"[10,0..3] := 0;
   "time"[10,4..5] := 500;
   "time"[10,6..25] := 0;
   "time"[11,0..3] := 0;
   "time"[11,4..5] := 500;
   "time"[11,6..25] := 0;
   "time"[12,0..3] := 0;
   "time"[12,4..5] := 500;
   "time"[12,6..25] := 0;
   "time"[13,0..3] := 0;
   "time"[13,4..5] := 500;
   "time"[13,6..25] := 0;
   "time"[14,0..3] := 0;
   "time"[14,4..5] := 500;
   "time"[14,6..25] := 0;
   "time"[15,0..25] := 0;
   "time"[16,0..3] := 0;
   "time"[16,4..5] := 500;
   "time"[16,6..25] := 0;
   "time"[17,0..3] := 0;
   "time"[17,4..5] := 500;
   "time"[17,6..25] := 0;
   "time"[18,0..3] := 0;
   "time"[18,4..5] := 500;
   "time"[18,6..25] := 0;
   "time"[19,0..3] := 0;
   "time"[19,4..5] := 500;
   "time"[19,6..25] := 0;
   "time"[20,0..25] := 0;
   "time"[21,0..25] := 0;
   "time"[22,0..25] := 0;
   "time"[23,0..25] := 0;
   "time"[24,0..25] := 0;
   "time"[25,0..25] := 0;
   "time"[26,0..25] := 0;
   "time"[27,0..25] := 0;
   "time"[28,0..25] := 0;
   "time"[29,0..25] := 0;
   "time"[30,0..25] := 0;
   "time"[31,0..25] := 0;
   "time"[32,0..25] := 0;
   number[0..2] := 8;
   number[3..6] := 6;
   number[7..14] := 9;
   number[15] := 8;
   number[16..19] := 9;
   number[20..32] := 0;
END_DATA_BLOCK

DATA_BLOCK "DB_MODEL"   // DB5
{ S7_Optimized_Access := 'TRUE' }
VERSION : 0.1
// stored: AutoNumber false, DBAccessibleFromOPCUA true, DBAccessibleFromWebserver true, IsOnlyStoredInLoadMemory false, IsRetainMemResEnabled false, IsWriteProtectedInAS false, MemoryReserve 100
   VAR RETAIN
      "name" : Array[0..32] of String[50];
   END_VAR
   VAR
      day : Int := 6;
      dayText : String := '    11';
      month : Int := 8;
      monthText : String := '     8';
      year : Int := 2012;
      yearReady : String := '2012';
      hour : Int := 17;
      hourText : String := '    17';
      minutes : Int := 30;
      minutesText : String := '    30';
      seconds : Int := 30;
      secondsText : String := '    31';
      active : Array[0..32] of Bool;
   END_VAR
   VAR RETAIN
      datum1 : Array[0..32] of String[50];
      datum2 : Array[0..32] of String[50];
      datum3 : Array[0..32] of String[50];
      datum4 : Array[0..32] of String[50];
      datum5 : Array[0..32] of String[50];
      datum6 : Array[0..32] of String[50];
      datum7 : Array[0..32] of String[50];
   END_VAR
BEGIN
   "name"[0] := 'RH MAN';
   "name"[1] := 'LH MAN';
   "name"[2] := 'RH MAN';
   "name"[3] := '721X';
   "name"[4] := 'STRAP';
   "name"[5] := 'BRACKET';
   "name"[6] := 'FULL FRAME';
   "name"[7..32] := '';
   active[0] := FALSE;
   active[1..6] := TRUE;
   active[7..32] := FALSE;
   datum1[0..2] := 'Z';
   datum1[3] := 'ddd';
   datum1[4..17] := 'Z';
   datum1[18..32] := '';
   datum2[0..17] := '410';
   datum2[18..32] := '';
   datum3[0..17] := '6';
   datum3[18..32] := '';
   datum4[0..2] := 'BACKREST W33A POWER MEMO L6';
   datum4[3] := 'prueba';
   datum4[4] := 'outter trackw33';
   datum4[5..16] := 'BACKREST W33A POWER MEMO L6';
   datum4[17] := 'P42LHNOMEM';
   datum4[18..32] := '';
   datum5[0] := '2389161X-01';
   datum5[1..2] := '2521784';
   datum5[3] := '2389161X-01';
   datum5[4..5] := '2282685X-01';
   datum5[6..16] := '2521784';
   datum5[17] := '2418723X-01';
   datum5[18..32] := '';
   datum6[0..32] := '';
   datum7[0..32] := '';
END_DATA_BLOCK

DATA_BLOCK "DB_INPUTS"   // DB1
{ S7_Optimized_Access := 'TRUE' }
VERSION : 0.1
// stored: AutoNumber false, DBAccessibleFromOPCUA true, DBAccessibleFromWebserver true, IsOnlyStoredInLoadMemory false, IsRetainMemResEnabled false, IsWriteProtectedInAS false, MemoryReserve 100
   VAR RETAIN
      intputSequence : Array[0..32, 0..25] of DInt;   // 32 entradas [modelo, paso]
   END_VAR
   VAR
      activeInputsReq : Array[0..31] of Bool;
   END_VAR
   VAR RETAIN
      maskSequence : Array[0..32, 0..25] of DInt;   // Máscara de entradas
   END_VAR
   VAR
      activeMask : Array[0..31] of Bool;
   END_VAR
   VAR RETAIN
      inputText : Array[0..31] of String;   // Texto HMI de cada entrada
   END_VAR
   VAR
      buttonStatus : Array[0..63] of Bool;
      activeInputsReqDInt : DInt := -2_130_444_284;   // Estado de sensores en directo
      inputActive : Array[0..31] of Bool;
      euchnerReading : Array[0..254] of Char;
      nestScannerReading : String := '';
      upperScannerReading : String := '';
      nestScanerReceived : Array[0..254] of Char;
      nestScanerReceivedString : String := '';
      upperScannerReceived : Array[0..254] of Char;
      upperScannerReceivedString : String := '';
      euchnerReadingString : String := '$01';
      laserReading : Word := 16#0000;
      laserConstant : Real := 0.0005802801;
      laserReadingInt : DInt := 0;
      readingConversion : LReal := 0.0;
      euchnerName : String := '';
      euchner : Array[0..257] of Byte;
   END_VAR
BEGIN
   intputSequence[0,0] := -2_130_444_283;
   intputSequence[0,1] := -1_996_150_012;
   intputSequence[0,2..4] := -2_146_096_376;
   intputSequence[0,5] := -2_130_367_736;
   intputSequence[0,6..7] := -2_130_367_740;
   intputSequence[0,8] := -2_130_444_284;
   intputSequence[0,9..25] := 0;
   intputSequence[1,0] := -2_130_444_283;
   intputSequence[1,1] := -1_996_082_428;
   intputSequence[1,2..3] := -2_142_358_768;
   intputSequence[1,4] := -2_142_358_640;
   intputSequence[1,5] := -2_142_358_652;
   intputSequence[1,6..7] := -2_130_300_156;
   intputSequence[1,8] := -2_130_444_284;
   intputSequence[1,9..25] := 0;
   intputSequence[2,0] := -2_130_444_283;
   intputSequence[2,1] := -1_996_150_012;
   intputSequence[2,2..4] := -2_146_096_376;
   intputSequence[2,5] := -2_130_367_736;
   intputSequence[2,6..7] := -2_130_367_740;
   intputSequence[2,8] := -2_130_444_284;
   intputSequence[2,9..25] := 0;
   intputSequence[3,0] := 84148229;
   intputSequence[3,1] := 1_057_235_716;
   intputSequence[3,2] := 1_175_724_802;
   intputSequence[3,3] := 101_720_834;
   intputSequence[3,4] := 101_982_978;
   intputSequence[3,5] := 84157188;
   intputSequence[3,6] := 84148228;
   intputSequence[3,7..25] := 0;
   intputSequence[4,0] := 84148229;
   intputSequence[4,1] := 1_057_236_740;
   intputSequence[4,2] := 1_175_725_826;
   intputSequence[4,3] := 101_721_858;
   intputSequence[4,4] := 101_984_002;
   intputSequence[4,5] := 84158212;
   intputSequence[4,6] := 84148228;
   intputSequence[4,7..25] := 0;
   intputSequence[5,0] := 84148229;
   intputSequence[5,1] := 1_057_284_868;
   intputSequence[5,2] := 1_175_773_954;
   intputSequence[5,3] := 101_769_986;
   intputSequence[5,4] := 102_032_130;
   intputSequence[5,5] := 84206340;
   intputSequence[5,6] := 84148228;
   intputSequence[5,7..25] := 0;
   intputSequence[6,0] := 84148229;
   intputSequence[6,1] := 1_057_285_892;
   intputSequence[6,2] := 1_175_774_978;
   intputSequence[6,3] := 101_771_010;
   intputSequence[6,4] := 102_033_154;
   intputSequence[6,5] := 84207364;
   intputSequence[6,6] := 84148228;
   intputSequence[6,7..25] := 0;
   intputSequence[7,0] := 23724868;
   intputSequence[7,1] := 827_780_422;
   intputSequence[7,2] := 44756294;
   intputSequence[7,3] := 44755974;
   intputSequence[7,4] := 1_252_650_334;
   intputSequence[7,5..7] := 1_118_432_670;
   intputSequence[7,8] := 1_118_432_414;
   intputSequence[7,9] := 44630336;
   intputSequence[7,10..25] := 0;
   intputSequence[8,0] := 23724353;
   intputSequence[8,1] := 827_776_326;
   intputSequence[8,2] := 44752198;
   intputSequence[8,3] := 44751878;
   intputSequence[8,4] := 1_252_646_238;
   intputSequence[8,5] := 1_118_428_574;
   intputSequence[8,6] := 1_118_428_318;
   intputSequence[8,7] := 1_118_428_574;
   intputSequence[8,8] := 1_118_428_318;
   intputSequence[8,9] := 44630336;
   intputSequence[8,10..25] := 0;
   intputSequence[9,0] := 321;
   intputSequence[9,1] := 4193656;
   intputSequence[9,2] := 2_017_459_576;
   intputSequence[9,3] := 1_077_935_482;
   intputSequence[9,4] := 1_073_745_282;
   intputSequence[9,5..6] := 1_073_745_538;
   intputSequence[9,7..9] := 320;
   intputSequence[9,10..25] := 0;
   intputSequence[10,0] := 321;
   intputSequence[10,1] := 4193656;
   intputSequence[10,2] := 2_017_459_576;
   intputSequence[10,3] := 1_077_935_482;
   intputSequence[10,4] := 1_073_745_282;
   intputSequence[10,5..6] := 1_073_745_538;
   intputSequence[10,7..9] := 320;
   intputSequence[10,10..25] := 0;
   intputSequence[11,0] := 321;
   intputSequence[11,1] := 4193656;
   intputSequence[11,2] := 2_017_459_576;
   intputSequence[11,3] := 1_077_935_482;
   intputSequence[11,4] := 1_073_745_282;
   intputSequence[11,5..6] := 1_073_745_538;
   intputSequence[11,7..9] := 320;
   intputSequence[11,10..25] := 0;
   intputSequence[12,0] := 321;
   intputSequence[12,1] := 8387960;
   intputSequence[12,2] := 2_021_653_880;
   intputSequence[12,3] := 1_082_129_786;
   intputSequence[12,4] := 1_077_939_586;
   intputSequence[12,5] := 1_077_939_842;
   intputSequence[12,6] := 1_073_745_538;
   intputSequence[12,7..9] := 320;
   intputSequence[12,10..25] := 0;
   intputSequence[13,0] := 321;
   intputSequence[13,1] := 4193656;
   intputSequence[13,2] := 2_017_459_576;
   intputSequence[13,3] := 1_077_935_482;
   intputSequence[13,4] := 1_073_745_282;
   intputSequence[13,5..6] := 1_073_745_538;
   intputSequence[13,7..9] := 320;
   intputSequence[13,10..25] := 0;
   intputSequence[14,0] := 321;
   intputSequence[14,1] := 4193656;
   intputSequence[14,2] := 2_017_459_576;
   intputSequence[14,3] := 1_077_935_482;
   intputSequence[14,4] := 1_073_745_282;
   intputSequence[14,5..6] := 1_073_745_538;
   intputSequence[14,7..9] := 320;
   intputSequence[14,10..25] := 0;
   intputSequence[15,0] := 11;
   intputSequence[15,1] := 63040522;
   intputSequence[15,2] := 1_338_108_938;
   intputSequence[15,3] := 65137674;
   intputSequence[15,4] := 65135628;
   intputSequence[15,5] := 65134612;
   intputSequence[15,6] := 57344;
   intputSequence[15,7] := 805_363_712;
   intputSequence[15,8] := 10;
   intputSequence[15,9..25] := 0;
   intputSequence[16,0] := 321;
   intputSequence[16,1] := 8387960;
   intputSequence[16,2] := 2_021_653_880;
   intputSequence[16,3] := 1_082_129_786;
   intputSequence[16,4] := 1_077_939_586;
   intputSequence[16,5] := 1_077_939_842;
   intputSequence[16,6] := 1_073_745_538;
   intputSequence[16,7..9] := 320;
   intputSequence[16,10..25] := 0;
   intputSequence[17,0] := 321;
   intputSequence[17,1] := 4193656;
   intputSequence[17,2] := 2_017_459_576;
   intputSequence[17,3] := 1_077_935_482;
   intputSequence[17,4] := 1_073_745_282;
   intputSequence[17,5..6] := 1_073_745_538;
   intputSequence[17,7..9] := 320;
   intputSequence[17,10..25] := 0;
   intputSequence[18,0] := 321;
   intputSequence[18,1] := 4193656;
   intputSequence[18,2] := 2_017_459_576;
   intputSequence[18,3] := 1_077_935_482;
   intputSequence[18,4] := 1_073_745_282;
   intputSequence[18,5..6] := 1_073_745_538;
   intputSequence[18,7..9] := 320;
   intputSequence[18,10..25] := 0;
   intputSequence[19,0] := 321;
   intputSequence[19,1] := 4193656;
   intputSequence[19,2] := 2_017_459_576;
   intputSequence[19,3] := 1_077_935_482;
   intputSequence[19,4] := 1_073_745_282;
   intputSequence[19,5..6] := 1_073_745_538;
   intputSequence[19,7..9] := 320;
   intputSequence[19,10..25] := 0;
   intputSequence[20,0..25] := 0;
   intputSequence[21,0..25] := 0;
   intputSequence[22,0..25] := 0;
   intputSequence[23,0..25] := 0;
   intputSequence[24,0..25] := 0;
   intputSequence[25,0..25] := 0;
   intputSequence[26,0..25] := 0;
   intputSequence[27,0..25] := 0;
   intputSequence[28,0..25] := 0;
   intputSequence[29,0..25] := 0;
   intputSequence[30,0..25] := 0;
   intputSequence[31,0..25] := 0;
   intputSequence[32,0..25] := 0;
   activeInputsReq[0] := TRUE;
   activeInputsReq[1] := FALSE;
   activeInputsReq[2] := TRUE;
   activeInputsReq[3..17] := FALSE;
   activeInputsReq[18] := TRUE;
   activeInputsReq[19..23] := FALSE;
   activeInputsReq[24] := TRUE;
   activeInputsReq[25..30] := FALSE;
   activeInputsReq[31] := TRUE;
   maskSequence[0,0] := 0;
   maskSequence[0,1] := 805_306_368;
   maskSequence[0,2] := 939_528_320;
   maskSequence[0,3] := 134_221_952;
   maskSequence[0,4] := 146_804_928;
   maskSequence[0,5] := 134_217_856;
   maskSequence[0,6..8] := 134_217_728;
   maskSequence[0,9..25] := 0;
   maskSequence[1,0] := 0;
   maskSequence[1,1] := 805_306_368;
   maskSequence[1,2] := 939_526_144;
   maskSequence[1,3..4] := 134_219_776;
   maskSequence[1,5] := 138_412_160;
   maskSequence[1,6] := 134_221_952;
   maskSequence[1,7..8] := 134_217_728;
   maskSequence[1,9..25] := 0;
   maskSequence[2,0] := 0;
   maskSequence[2,1] := 805_306_368;
   maskSequence[2,2] := 939_528_320;
   maskSequence[2,3] := 134_221_952;
   maskSequence[2,4] := 146_804_928;
   maskSequence[2,5] := 134_217_856;
   maskSequence[2,6..8] := 134_217_728;
   maskSequence[2,9..25] := 0;
   maskSequence[3,0] := 0;
   maskSequence[3,1] := 202752;
   maskSequence[3,2] := 948_115_456;
   maskSequence[3,3] := 2_055_411_712;
   maskSequence[3,4] := 998_447_104;
   maskSequence[3,5] := 948_115_456;
   maskSequence[3,6] := 939_726_848;
   maskSequence[3,7..25] := 0;
   maskSequence[4,0] := 0;
   maskSequence[4,1] := 202752;
   maskSequence[4,2] := 948_115_456;
   maskSequence[4,3] := 2_055_411_712;
   maskSequence[4,4] := 998_447_104;
   maskSequence[4,5] := 948_115_456;
   maskSequence[4,6] := 939_726_848;
   maskSequence[4,7..25] := 0;
   maskSequence[5,0] := 0;
   maskSequence[5,1] := 202752;
   maskSequence[5,2] := 948_115_456;
   maskSequence[5,3] := 2_055_411_712;
   maskSequence[5,4] := 998_447_104;
   maskSequence[5,5] := 948_115_456;
   maskSequence[5,6] := 939_726_848;
   maskSequence[5,7..25] := 0;
   maskSequence[6,0] := 0;
   maskSequence[6,1] := 202752;
   maskSequence[6,2] := 948_115_456;
   maskSequence[6,3] := 2_055_411_712;
   maskSequence[6,4] := 998_447_104;
   maskSequence[6,5] := 948_115_456;
   maskSequence[6,6] := 939_726_848;
   maskSequence[6,7..25] := 0;
   maskSequence[7,0] := 66848767;
   maskSequence[7,1] := 66846720;
   maskSequence[7,2..3] := 66847168;
   maskSequence[7,4..6] := 66846720;
   maskSequence[7,7] := 66846976;
   maskSequence[7,8] := 66846720;
   maskSequence[7,9] := 66847168;
   maskSequence[7,10..25] := 0;
   maskSequence[8,0..1] := 66846720;
   maskSequence[8,2..3] := 66847168;
   maskSequence[8,4..5] := 66846720;
   maskSequence[8,6..7] := 66846976;
   maskSequence[8,8] := 66846720;
   maskSequence[8,9] := 66847168;
   maskSequence[8,10..25] := 0;
   maskSequence[9,0] := -322;
   maskSequence[9,1] := 2_014_248_960;
   maskSequence[9,2..3] := 983040;
   maskSequence[9,4..5] := 79687736;
   maskSequence[9,6] := 134_213_948;
   maskSequence[9,7..8] := -2;
   maskSequence[9,9] := 134_217_406;
   maskSequence[9,10..25] := 0;
   maskSequence[10,0] := -322;
   maskSequence[10,1] := 2_014_289_920;
   maskSequence[10,2..3] := 1024000;
   maskSequence[10,4..5] := 79687736;
   maskSequence[10,6] := 134_213_948;
   maskSequence[10,7..8] := -2;
   maskSequence[10,9] := 134_217_406;
   maskSequence[10,10..25] := 0;
   maskSequence[11,0] := -322;
   maskSequence[11,1] := 2_014_248_960;
   maskSequence[11,2..3] := 983040;
   maskSequence[11,4..5] := 79687736;
   maskSequence[11,6] := 134_213_948;
   maskSequence[11,7..8] := -2;
   maskSequence[11,9] := 134_217_406;
   maskSequence[11,10..25] := 0;
   maskSequence[12,0] := -322;
   maskSequence[12,1] := 2_014_248_960;
   maskSequence[12,2..3] := 983040;
   maskSequence[12,4..5] := 79687736;
   maskSequence[12,6] := 134_213_948;
   maskSequence[12,7..8] := -2;
   maskSequence[12,9] := 134_217_406;
   maskSequence[12,10..25] := 0;
   maskSequence[13,0] := -322;
   maskSequence[13,1] := 2_014_248_960;
   maskSequence[13,2..3] := 983040;
   maskSequence[13,4..5] := 79687736;
   maskSequence[13,6] := 134_213_948;
   maskSequence[13,7..8] := -2;
   maskSequence[13,9] := 134_217_406;
   maskSequence[13,10..25] := 0;
   maskSequence[14,0] := -322;
   maskSequence[14,1] := 2_014_248_960;
   maskSequence[14,2] := 806_289_408;
   maskSequence[14,3] := 983040;
   maskSequence[14,4..5] := 79687736;
   maskSequence[14,6] := 134_213_948;
   maskSequence[14,7..8] := -2;
   maskSequence[14,9] := 134_217_406;
   maskSequence[14,10..25] := 0;
   maskSequence[15,0] := 0;
   maskSequence[15,1] := 2_080_374_784;
   maskSequence[15,2..3] := 805_306_368;
   maskSequence[15,4..5] := 868_220_928;
   maskSequence[15,6..7] := 268_435_452;
   maskSequence[15,8..25] := 0;
   maskSequence[16,0] := -322;
   maskSequence[16,1] := 2_014_248_960;
   maskSequence[16,2..3] := 983040;
   maskSequence[16,4..5] := 79687736;
   maskSequence[16,6] := 134_213_948;
   maskSequence[16,7..8] := -2;
   maskSequence[16,9] := 134_217_406;
   maskSequence[16,10..25] := 0;
   maskSequence[17,0] := -322;
   maskSequence[17,1] := 2_014_248_960;
   maskSequence[17,2..3] := 983040;
   maskSequence[17,4..5] := 79687736;
   maskSequence[17,6] := 134_213_948;
   maskSequence[17,7..8] := -2;
   maskSequence[17,9] := 134_217_406;
   maskSequence[17,10..25] := 0;
   maskSequence[18,0] := -322;
   maskSequence[18,1] := 2_014_248_960;
   maskSequence[18,2..3] := 983040;
   maskSequence[18,4..5] := 79687736;
   maskSequence[18,6] := 134_213_948;
   maskSequence[18,7..8] := -2;
   maskSequence[18,9] := 134_217_406;
   maskSequence[18,10..25] := 0;
   maskSequence[19,0] := -322;
   maskSequence[19,1] := 2_014_248_960;
   maskSequence[19,2..3] := 983040;
   maskSequence[19,4..5] := 79687736;
   maskSequence[19,6] := 134_213_948;
   maskSequence[19,7..8] := -2;
   maskSequence[19,9] := 134_217_406;
   maskSequence[19,10..25] := 0;
   maskSequence[20,0..25] := 0;
   maskSequence[21,0..25] := 0;
   maskSequence[22,0..25] := 0;
   maskSequence[23,0..25] := 0;
   maskSequence[24,0..25] := 0;
   maskSequence[25,0..25] := 0;
   maskSequence[26,0..25] := 0;
   maskSequence[27,0..25] := 0;
   maskSequence[28,0..25] := 0;
   maskSequence[29,0..25] := 0;
   maskSequence[30,0..25] := 0;
   maskSequence[31,0..25] := 0;
   maskSequence[32,0..25] := 0;
   activeMask[0..31] := FALSE;
   inputText[0] := 'CLEAR DATA';
   inputText[1] := 'LEFT TOOLING WORK POS';
   inputText[2] := 'LEFTTOOLING HOME POS';
   inputText[3] := 'LEFT TOOLING POS 1';
   inputText[4] := 'LEFT TOOOLLING POS 3';
   inputText[5] := 'LEFT TOOLING POS 2';
   inputText[6] := 'LEFT INSERTIONN EXT NOK';
   inputText[7] := 'LEFT INSERTIONN EXT OK';
   inputText[8] := 'PRODUCT INSERTED LH';
   inputText[9] := 'PRODUCT INSERTED RH';
   inputText[10] := 'STRAP DETECTION';
   inputText[11] := 'LEFT MANUAL FRAME PRES';
   inputText[12] := 'RIGHT MANUAL FRAME PRES';
   inputText[13] := 'FRAME PRES';
   inputText[14] := 'LEFTT BRACKET DETECTION';
   inputText[15] := 'RIGHT BRACKET DETECTION';
   inputText[16] := 'LEFT COLOR SPRING';
   inputText[17] := 'RIGHT COLOR SPRING';
   inputText[18] := 'TORQUE TOOLING HOME';
   inputText[19] := 'RIGHT TOOLING POS 1';
   inputText[20] := 'RIGHT TOOLING POS 3';
   inputText[21] := 'RIGHT TOOLING POS 2';
   inputText[22] := 'RIGHT INSERTION EXT OK';
   inputText[23] := 'RIGHT INSERTION EXTNOK';
   inputText[24] := 'RIGHT TOOLING HOME';
   inputText[25] := 'WASHER INSERTED';
   inputText[26] := 'POWER TOOLING';
   inputText[27] := 'NEST SCANNER';
   inputText[28] := 'ANGLE SCANNER';
   inputText[29] := 'UPPER SCANNER LABEL1';
   inputText[30] := 'UPPER SCANNER LABEL 2';
   inputText[31] := 'MANUAL TOOLING';
   buttonStatus[0..2] := FALSE;
   buttonStatus[3] := TRUE;
   buttonStatus[4..7] := FALSE;
   buttonStatus[8..9] := TRUE;
   buttonStatus[10] := FALSE;
   buttonStatus[11] := TRUE;
   buttonStatus[12] := FALSE;
   buttonStatus[13] := TRUE;
   buttonStatus[14..15] := FALSE;
   buttonStatus[16] := TRUE;
   buttonStatus[17] := FALSE;
   buttonStatus[18] := TRUE;
   buttonStatus[19] := FALSE;
   buttonStatus[20] := TRUE;
   buttonStatus[21..30] := FALSE;
   buttonStatus[31] := TRUE;
   buttonStatus[32..38] := FALSE;
   buttonStatus[39] := TRUE;
   buttonStatus[40..43] := FALSE;
   buttonStatus[44] := TRUE;
   buttonStatus[45..58] := FALSE;
   buttonStatus[59] := TRUE;
   buttonStatus[60..63] := FALSE;
   inputActive[0..1] := FALSE;
   inputActive[2] := TRUE;
   inputActive[3..7] := FALSE;
   inputActive[8..9] := TRUE;
   inputActive[10] := FALSE;
   inputActive[11..13] := TRUE;
   inputActive[14..16] := FALSE;
   inputActive[17..18] := TRUE;
   inputActive[19..23] := FALSE;
   inputActive[24] := TRUE;
   inputActive[25..30] := FALSE;
   inputActive[31] := TRUE;
   euchnerReading[0] := '$01';
   euchnerReading[1..127] := '$00';
   euchnerReading[128..254] := ' ';
   nestScanerReceived[0..254] := ' ';
   upperScannerReceived[0..254] := ' ';
   euchner[0..1] := 16#00;
   euchner[2] := 16#44;
   euchner[3..7] := 16#00;
   euchner[8..147] := 16#20;
   euchner[148..257] := 16#00;
END_DATA_BLOCK

DATA_BLOCK "DB_Outputs"   // DB2
{ S7_Optimized_Access := 'TRUE' }
VERSION : 0.1
// stored: AutoNumber false, DBAccessibleFromOPCUA true, DBAccessibleFromWebserver true, IsOnlyStoredInLoadMemory false, IsRetainMemResEnabled false, IsWriteProtectedInAS false, MemoryReserve 0
   VAR RETAIN
      outputSequence : Array[0..32, 0..25] of DInt;   // 32 salidas [modelo, paso]
   END_VAR
   VAR
      activeOutputsReq : Array[0..31] of Bool;
   END_VAR
   VAR RETAIN
      maskSequence : Array[0..32, 0..25] of DInt;   // Máscara de salidas
   END_VAR
   VAR
      activeMask : Array[0..31] of Bool;
      active : DInt := 8362;
      outputsActive : Array[0..31] of Bool;
      text : Array[0..31] of String;   // Texto HMI de cada salida
      availableNameManipulate : Array[0..8] of String;   // Texto HMI en pagina Manual
      status : Array[0..63] of Bool;
      cylinderDirectionA : Array[0..9] of Bool;   // Variable HMI para activar avance
      cylinderDirectionB : Array[0..9] of Bool;   // Variable HMI para activar retroceso
      cylinderDirectionAActive : Array[0..9] of Bool;   // Variable HMI para enclavamiento avance
      cylinderDirectionBActive : Array[0..9] of Bool;   // Variable HMI para enclavamiento retroceso
      cylinderDirectionAStatus : Array[0..9] of Bool;   // Variable HMI para enclavamiento avance
      cylinderDirectionBStatus : Array[0..9] of Bool;   // Variable HMI para enclavamiento retroceso
      vent : Array[0..9] of Bool;   // Variable HMI para desactivar electroválvula
      "ESTADO DISP MANIPULAR" : Array[0..9] of Int;   // Variable HMI para estado de los botones de manipulación
      activateOutput : Array[0..31] of Bool;
      activeAlarm : Bool := FALSE;
      showTextOutPuts : Bool := FALSE;
      cicleTime : Int := 0;
      cicleTimeTimerReset : Bool := FALSE;
      timer1 { S7_SetPoint := 'True'} : TON_TIME;
      timer2 { S7_SetPoint := 'True'} : TON_TIME;
      timer3 { S7_SetPoint := 'True'} : TON_TIME;
      timer4 { S7_SetPoint := 'True'} : TON_TIME;
      timer5 { S7_SetPoint := 'True'} : TON_TIME;
      timer6 { S7_SetPoint := 'True'} : TON_TIME;
      timer7 { S7_SetPoint := 'True'} : TON_TIME;
      timer8 { S7_SetPoint := 'True'} : TON_TIME;
      timer9 { S7_SetPoint := 'True'} : TON_TIME;
      timer10 { S7_SetPoint := 'True'} : TON_TIME;
      timer11 { S7_SetPoint := 'True'} : TON_TIME;
      timer12 { S7_SetPoint := 'True'} : TON_TIME;
      timer13 { S7_SetPoint := 'True'} : TON_TIME;
      timer14 { S7_SetPoint := 'True'} : TON_TIME;
      timer15 { S7_SetPoint := 'True'} : TON_TIME;
      timer16 { S7_SetPoint := 'True'} : TON_TIME;
      timer17 { S7_SetPoint := 'True'} : TON_TIME;
      timer18 { S7_SetPoint := 'True'} : TON_TIME;
      timer19 { S7_SetPoint := 'True'} : TON_TIME;
      timer20 { S7_SetPoint := 'True'} : TON_TIME;
      timer21 { S7_SetPoint := 'True'} : TON_TIME;
      timer22 { S7_SetPoint := 'True'} : TON_TIME;
      timer23 { S7_SetPoint := 'True'} : TON_TIME;
      timer24 { S7_SetPoint := 'True'} : TON_TIME;
      timer25 { S7_SetPoint := 'True'} : TON_TIME;
      timer26 { S7_SetPoint := 'True'} : TON_TIME;
      timer27 { S7_SetPoint := 'True'} : TON_TIME;
      timer28 { S7_SetPoint := 'True'} : TON_TIME;
      timer29 { S7_SetPoint := 'True'} : TON_TIME;
      timer30 { S7_SetPoint := 'True'} : TON_TIME;
      timer31 { S7_SetPoint := 'True'} : TON_TIME;
      "timer" { S7_SetPoint := 'True'} : Array[0..31] of ton_time;
      reset : Bool := FALSE;
      timerReset : Bool := FALSE;
      visibility : Array[0..8] of Bool;
      visualizeCicleTime : Int := 90;
      scannerOk : Array[0..5] of Bool;
      scannerLength : Array[0..5] of Int;
      cilinder1 : Bool := TRUE;
      cilinder2 : Bool := TRUE;
      cilinder3 : Bool := TRUE;
      cilinder4 : Bool := FALSE;
      cilinder5 : Bool := FALSE;
      cilinder6 : Bool := FALSE;
      cilinder7 : Bool := FALSE;
      cilinder8 : Bool := FALSE;
   END_VAR
BEGIN
   outputSequence[0,0] := 8362;
   outputSequence[0,1] := 8353;
   outputSequence[0,2] := 4265;
   outputSequence[0,3] := 4197;
   outputSequence[0,4] := 4181;
   outputSequence[0,5] := 4201;
   outputSequence[0,6..8] := 8361;
   outputSequence[0,9..25] := 0;
   outputSequence[1,0] := 8362;
   outputSequence[1,1] := 8293;
   outputSequence[1,2] := 8345;
   outputSequence[1,3] := 8277;
   outputSequence[1,4] := 4181;
   outputSequence[1,5] := 8341;
   outputSequence[1,6..8] := 8361;
   outputSequence[1,9..25] := 0;
   outputSequence[2,0] := 8362;
   outputSequence[2,1] := 8353;
   outputSequence[2,2] := 4265;
   outputSequence[2,3] := 4197;
   outputSequence[2,4] := 4181;
   outputSequence[2,5] := 4201;
   outputSequence[2,6..8] := 8361;
   outputSequence[2,9..25] := 0;
   outputSequence[3,0] := 8362;
   outputSequence[3,1] := 8293;
   outputSequence[3,2] := 8361;
   outputSequence[3,3] := 1_073_746_006;
   outputSequence[3,4] := 4181;
   outputSequence[3,5] := 8361;
   outputSequence[3,6] := 8293;
   outputSequence[3,7..25] := 0;
   outputSequence[4,0] := 8362;
   outputSequence[4,1] := 8293;
   outputSequence[4,2] := 8361;
   outputSequence[4,3] := 1_073_746_006;
   outputSequence[4,4] := 4181;
   outputSequence[4,5] := 8361;
   outputSequence[4,6] := 8293;
   outputSequence[4,7..25] := 0;
   outputSequence[5,0] := 8362;
   outputSequence[5,1] := 8293;
   outputSequence[5,2] := 8361;
   outputSequence[5,3] := 1_073_746_006;
   outputSequence[5,4] := 4181;
   outputSequence[5,5] := 8361;
   outputSequence[5,6] := 8293;
   outputSequence[5,7..25] := 0;
   outputSequence[6,0] := 8362;
   outputSequence[6,1] := 8293;
   outputSequence[6,2] := 8361;
   outputSequence[6,3] := 1_073_746_006;
   outputSequence[6,4] := 4181;
   outputSequence[6,5] := 8361;
   outputSequence[6,6] := 8293;
   outputSequence[6,7..25] := 0;
   outputSequence[7,0] := 90;
   outputSequence[7,1] := 85;
   outputSequence[7,2] := 170;
   outputSequence[7,3] := 938;
   outputSequence[7,4] := 170;
   outputSequence[7,5] := 66726;
   outputSequence[7,6] := 170;
   outputSequence[7,7] := 169;
   outputSequence[7,8] := 133289;
   outputSequence[7,9] := 89;
   outputSequence[7,10..25] := 0;
   outputSequence[8,0] := 90;
   outputSequence[8,1] := 85;
   outputSequence[8,2] := 170;
   outputSequence[8,3] := 938;
   outputSequence[8,4] := 170;
   outputSequence[8,5] := 66726;
   outputSequence[8,6] := 170;
   outputSequence[8,7] := 169;
   outputSequence[8,8] := 133289;
   outputSequence[8,9] := 89;
   outputSequence[8,10..25] := 0;
   outputSequence[9,0] := 336;
   outputSequence[9,1] := 298;
   outputSequence[9,2] := 299;
   outputSequence[9,3] := 171;
   outputSequence[9,4] := 65715;
   outputSequence[9,5] := 65739;
   outputSequence[9,6] := 171;
   outputSequence[9,7] := 301;
   outputSequence[9,8] := 134_742_317;
   outputSequence[9,9] := 341;
   outputSequence[9,10..25] := 0;
   outputSequence[10,0] := 336;
   outputSequence[10,1] := 298;
   outputSequence[10,2] := 299;
   outputSequence[10,3] := 171;
   outputSequence[10,4] := 65715;
   outputSequence[10,5] := 65739;
   outputSequence[10,6] := 171;
   outputSequence[10,7] := 301;
   outputSequence[10,8] := 134_742_317;
   outputSequence[10,9] := 341;
   outputSequence[10,10..25] := 0;
   outputSequence[11,0] := 336;
   outputSequence[11,1] := 298;
   outputSequence[11,2] := 299;
   outputSequence[11,3] := 171;
   outputSequence[11,4] := 65715;
   outputSequence[11,5] := 65739;
   outputSequence[11,6] := 171;
   outputSequence[11,7] := 301;
   outputSequence[11,8] := 134_742_317;
   outputSequence[11,9] := 341;
   outputSequence[11,10..25] := 0;
   outputSequence[12,0] := 336;
   outputSequence[12,1] := 298;
   outputSequence[12,2] := 299;
   outputSequence[12,3] := 171;
   outputSequence[12,4] := 65715;
   outputSequence[12,5] := 65739;
   outputSequence[12,6] := 171;
   outputSequence[12,7] := 301;
   outputSequence[12,8] := 134_742_317;
   outputSequence[12,9] := 341;
   outputSequence[12,10..25] := 0;
   outputSequence[13,0] := 336;
   outputSequence[13,1] := 298;
   outputSequence[13,2] := 299;
   outputSequence[13,3] := 171;
   outputSequence[13,4] := 65715;
   outputSequence[13,5] := 65739;
   outputSequence[13,6] := 171;
   outputSequence[13,7] := 301;
   outputSequence[13,8] := 134_742_317;
   outputSequence[13,9] := 341;
   outputSequence[13,10..25] := 0;
   outputSequence[14,0] := 336;
   outputSequence[14,1] := 117_440_810;
   outputSequence[14,2] := 299;
   outputSequence[14,3] := 171;
   outputSequence[14,4] := 65715;
   outputSequence[14,5] := 65739;
   outputSequence[14,6] := 171;
   outputSequence[14,7] := 301;
   outputSequence[14,8] := 134_742_317;
   outputSequence[14,9] := 341;
   outputSequence[14,10..25] := 0;
   outputSequence[15,0] := 5408;
   outputSequence[15,1..2] := 4768;
   outputSequence[15,3] := 800;
   outputSequence[15,4] := 11040;
   outputSequence[15,5] := 11424;
   outputSequence[15,6] := 4800;
   outputSequence[15,7] := 37568;
   outputSequence[15,8] := 5440;
   outputSequence[15,9..25] := 0;
   outputSequence[16,0] := 336;
   outputSequence[16,1] := 298;
   outputSequence[16,2] := 299;
   outputSequence[16,3] := 171;
   outputSequence[16,4] := 65715;
   outputSequence[16,5] := 65739;
   outputSequence[16,6] := 171;
   outputSequence[16,7] := 301;
   outputSequence[16,8] := 134_742_317;
   outputSequence[16,9] := 341;
   outputSequence[16,10..25] := 0;
   outputSequence[17,0] := 336;
   outputSequence[17,1] := 298;
   outputSequence[17,2] := 299;
   outputSequence[17,3] := 171;
   outputSequence[17,4] := 65715;
   outputSequence[17,5] := 65739;
   outputSequence[17,6] := 171;
   outputSequence[17,7] := 301;
   outputSequence[17,8] := 134_742_317;
   outputSequence[17,9] := 341;
   outputSequence[17,10..25] := 0;
   outputSequence[18,0] := 336;
   outputSequence[18,1] := 117_440_810;
   outputSequence[18,2] := 117_440_811;
   outputSequence[18,3] := 171;
   outputSequence[18,4] := 65715;
   outputSequence[18,5] := 65739;
   outputSequence[18,6] := 171;
   outputSequence[18,7] := 301;
   outputSequence[18,8] := 940_048_685;
   outputSequence[18,9] := 341;
   outputSequence[18,10..25] := 0;
   outputSequence[19,0] := 336;
   outputSequence[19,1] := 298;
   outputSequence[19,2] := 299;
   outputSequence[19,3] := 171;
   outputSequence[19,4] := 65715;
   outputSequence[19,5] := 65739;
   outputSequence[19,6] := 171;
   outputSequence[19,7] := 301;
   outputSequence[19,8] := 134_742_317;
   outputSequence[19,9] := 341;
   outputSequence[19,10..25] := 0;
   outputSequence[20,0..25] := 0;
   outputSequence[21,0..25] := 0;
   outputSequence[22,0..25] := 0;
   outputSequence[23,0..25] := 0;
   outputSequence[24,0..25] := 0;
   outputSequence[25,0..25] := 0;
   outputSequence[26,0..25] := 0;
   outputSequence[27,0..25] := 0;
   outputSequence[28,0..25] := 0;
   outputSequence[29,0..25] := 0;
   outputSequence[30,0..25] := 0;
   outputSequence[31,0..25] := 0;
   outputSequence[32,0..25] := 0;
   activeOutputsReq[0] := FALSE;
   activeOutputsReq[1] := TRUE;
   activeOutputsReq[2] := FALSE;
   activeOutputsReq[3] := TRUE;
   activeOutputsReq[4] := FALSE;
   activeOutputsReq[5] := TRUE;
   activeOutputsReq[6] := FALSE;
   activeOutputsReq[7] := TRUE;
   activeOutputsReq[8..12] := FALSE;
   activeOutputsReq[13] := TRUE;
   activeOutputsReq[14..31] := FALSE;
   maskSequence[0,0..3] := 0;
   maskSequence[0,4] := 4112;
   maskSequence[0,5..25] := 0;
   maskSequence[1,0..3] := 0;
   maskSequence[1,4] := 4096;
   maskSequence[1,5..25] := 0;
   maskSequence[2,0..3] := 0;
   maskSequence[2,4] := 4112;
   maskSequence[2,5..25] := 0;
   maskSequence[3,0..3] := 0;
   maskSequence[3,4..6] := 1_073_741_824;
   maskSequence[3,7..25] := 0;
   maskSequence[4,0..3] := 0;
   maskSequence[4,4..6] := 1_073_741_824;
   maskSequence[4,7..25] := 0;
   maskSequence[5,0..3] := 0;
   maskSequence[5,4..6] := 1_073_741_824;
   maskSequence[5,7..25] := 0;
   maskSequence[6,0..3] := 0;
   maskSequence[6,4..6] := 1_073_741_824;
   maskSequence[6,7..25] := 0;
   maskSequence[7,0..25] := 0;
   maskSequence[8,0..25] := 0;
   maskSequence[9,0] := 6;
   maskSequence[9,1..4] := 8;
   maskSequence[9,5] := 32768;
   maskSequence[9,6] := 10;
   maskSequence[9,7] := -134_283_256;
   maskSequence[9,8] := -134_742_017;
   maskSequence[9,9..25] := 0;
   maskSequence[10,0] := 6;
   maskSequence[10,1..4] := 8;
   maskSequence[10,5] := 32768;
   maskSequence[10,6] := 10;
   maskSequence[10,7] := -134_283_256;
   maskSequence[10,8] := -134_742_017;
   maskSequence[10,9..25] := 0;
   maskSequence[11,0] := 6;
   maskSequence[11,1..4] := 8;
   maskSequence[11,5] := 32768;
   maskSequence[11,6] := 10;
   maskSequence[11,7] := -134_283_256;
   maskSequence[11,8] := -134_742_017;
   maskSequence[11,9..25] := 0;
   maskSequence[12,0] := 6;
   maskSequence[12,1..4] := 8;
   maskSequence[12,5] := 32768;
   maskSequence[12,6] := 10;
   maskSequence[12,7] := -134_283_256;
   maskSequence[12,8] := -134_742_017;
   maskSequence[12,9..25] := 0;
   maskSequence[13,0] := 6;
   maskSequence[13,1..4] := 8;
   maskSequence[13,5] := 32768;
   maskSequence[13,6] := 10;
   maskSequence[13,7] := -134_283_256;
   maskSequence[13,8] := -134_742_017;
   maskSequence[13,9..25] := 0;
   maskSequence[14,0] := 6;
   maskSequence[14,1..4] := 8;
   maskSequence[14,5] := 32768;
   maskSequence[14,6] := 10;
   maskSequence[14,7] := -134_283_256;
   maskSequence[14,8] := -134_742_017;
   maskSequence[14,9..25] := 0;
   maskSequence[15,0] := 4096;
   maskSequence[15,1..2] := 0;
   maskSequence[15,3] := 32;
   maskSequence[15,4..25] := 0;
   maskSequence[16,0] := 6;
   maskSequence[16,1..4] := 8;
   maskSequence[16,5] := 32768;
   maskSequence[16,6] := 10;
   maskSequence[16,7] := -134_283_256;
   maskSequence[16,8] := -134_742_017;
   maskSequence[16,9..25] := 0;
   maskSequence[17,0] := 6;
   maskSequence[17,1..4] := 8;
   maskSequence[17,5] := 32768;
   maskSequence[17,6] := 10;
   maskSequence[17,7] := -134_283_256;
   maskSequence[17,8] := -134_742_017;
   maskSequence[17,9..25] := 0;
   maskSequence[18,0] := 117_440_518;
   maskSequence[18,1..2] := 8;
   maskSequence[18,3..4] := 117_440_520;
   maskSequence[18,5] := 117_473_280;
   maskSequence[18,6] := 117_440_522;
   maskSequence[18,7] := -134_283_256;
   maskSequence[18,8] := -940_048_385;
   maskSequence[18,9] := 117_440_512;
   maskSequence[18,10..25] := 0;
   maskSequence[19,0] := 6;
   maskSequence[19,1..4] := 8;
   maskSequence[19,5] := 32768;
   maskSequence[19,6] := 10;
   maskSequence[19,7] := -134_283_256;
   maskSequence[19,8] := -134_742_017;
   maskSequence[19,9..25] := 0;
   maskSequence[20,0..25] := 0;
   maskSequence[21,0..25] := 0;
   maskSequence[22,0..25] := 0;
   maskSequence[23,0..25] := 0;
   maskSequence[24,0..25] := 0;
   maskSequence[25,0..25] := 0;
   maskSequence[26,0..25] := 0;
   maskSequence[27,0..25] := 0;
   maskSequence[28,0..25] := 0;
   maskSequence[29,0..25] := 0;
   maskSequence[30,0..25] := 0;
   maskSequence[31,0..25] := 0;
   maskSequence[32,0..25] := 0;
   activeMask[0..31] := FALSE;
   outputsActive[0] := FALSE;
   outputsActive[1] := TRUE;
   outputsActive[2] := FALSE;
   outputsActive[3] := TRUE;
   outputsActive[4] := FALSE;
   outputsActive[5] := TRUE;
   outputsActive[6] := FALSE;
   outputsActive[7] := TRUE;
   outputsActive[8..12] := FALSE;
   outputsActive[13] := TRUE;
   outputsActive[14..31] := FALSE;
   text[0] := 'Torque Tooling Lock CYL  EXT';
   text[1] := 'Torque Toooling Lock CYL RET';
   text[2] := 'Right Tooling Lock CYL EXT';
   text[3] := 'Right Tooing Lock CYL RET';
   text[4] := 'Right MAN Rod Ins EXT';
   text[5] := 'Right MAN Rod Ins RET';
   text[6] := 'Left Tooling Lock EXT';
   text[7] := 'Left Tooling Lock RET';
   text[8..11] := 'SPARE';
   text[12] := 'Left Insertion CYLS EXT';
   text[13] := 'Left Insertion CYLS RET';
   text[14..15] := 'RESERVA';
   text[16..29] := 'SPARE';
   text[30] := 'Torque';
   text[31] := 'SPARE';
   availableNameManipulate[0] := 'Bloqueo Tooling Izq';
   availableNameManipulate[1] := 'Bloqueo TooIing Der';
   availableNameManipulate[2] := 'Bloqueo Tooling Torque';
   availableNameManipulate[3] := 'Insercion RH';
   availableNameManipulate[4] := 'Insercion LH';
   availableNameManipulate[5] := 'Spare 5';
   availableNameManipulate[6..8] := '';
   status[0] := TRUE;
   status[1] := FALSE;
   status[2] := TRUE;
   status[3..4] := FALSE;
   status[5..6] := TRUE;
   status[7..11] := FALSE;
   status[12] := TRUE;
   status[13..63] := FALSE;
   cylinderDirectionA[0..9] := FALSE;
   cylinderDirectionB[0..9] := FALSE;
   cylinderDirectionAActive[0..9] := FALSE;
   cylinderDirectionBActive[0..2] := TRUE;
   cylinderDirectionBActive[3..5] := FALSE;
   cylinderDirectionBActive[6] := TRUE;
   cylinderDirectionBActive[7..9] := FALSE;
   cylinderDirectionAStatus[0..9] := FALSE;
   cylinderDirectionBStatus[0..9] := FALSE;
   vent[0..9] := FALSE;
   "ESTADO DISP MANIPULAR"[0..9] := 0;
   activateOutput[0] := FALSE;
   activateOutput[1] := TRUE;
   activateOutput[2] := FALSE;
   activateOutput[3] := TRUE;
   activateOutput[4] := FALSE;
   activateOutput[5] := TRUE;
   activateOutput[6] := FALSE;
   activateOutput[7] := TRUE;
   activateOutput[8..12] := FALSE;
   activateOutput[13] := TRUE;
   activateOutput[14..31] := FALSE;
   timer1.PT := T#0MS;
   timer1.IN := FALSE;
   timer2.PT := T#0MS;
   timer2.IN := FALSE;
   timer3.PT := T#0MS;
   timer3.IN := FALSE;
   timer4.PT := T#0MS;
   timer4.IN := FALSE;
   timer5.PT := T#0MS;
   timer5.IN := FALSE;
   timer6.PT := T#0MS;
   timer6.IN := FALSE;
   timer7.PT := T#0MS;
   timer7.IN := FALSE;
   timer8.PT := T#0MS;
   timer8.IN := FALSE;
   timer9.PT := T#0MS;
   timer9.IN := FALSE;
   timer10.PT := T#0MS;
   timer10.IN := FALSE;
   timer11.PT := T#0MS;
   timer11.IN := FALSE;
   timer12.PT := T#0MS;
   timer12.IN := FALSE;
   timer13.PT := T#0MS;
   timer13.IN := FALSE;
   timer14.PT := T#0MS;
   timer14.IN := FALSE;
   timer15.PT := T#0MS;
   timer15.IN := FALSE;
   timer16.PT := T#0MS;
   timer16.IN := FALSE;
   timer17.PT := T#0MS;
   timer17.IN := FALSE;
   timer18.PT := T#0MS;
   timer18.IN := FALSE;
   timer19.PT := T#0MS;
   timer19.IN := FALSE;
   timer20.PT := T#0MS;
   timer20.IN := FALSE;
   timer21.PT := T#0MS;
   timer21.IN := FALSE;
   timer22.PT := T#0MS;
   timer22.IN := FALSE;
   timer23.PT := T#0MS;
   timer23.IN := FALSE;
   timer24.PT := T#0MS;
   timer24.IN := FALSE;
   timer25.PT := T#0MS;
   timer25.IN := FALSE;
   timer26.PT := T#0MS;
   timer26.IN := FALSE;
   timer27.PT := T#0MS;
   timer27.IN := FALSE;
   timer28.PT := T#0MS;
   timer28.IN := FALSE;
   timer29.PT := T#0MS;
   timer29.IN := FALSE;
   timer30.PT := T#0MS;
   timer30.IN := FALSE;
   timer31.PT := T#0MS;
   timer31.IN := FALSE;
   "timer"[0..31].PT := T#0MS;
   "timer"[0..31].IN := FALSE;
   visibility[0] := FALSE;
   visibility[1..3] := TRUE;
   visibility[4..8] := FALSE;
   scannerOk[0..5] := FALSE;
   scannerLength[0] := 0;
   scannerLength[1..3] := 3;
   scannerLength[4..5] := 0;
END_DATA_BLOCK

DATA_BLOCK "ALARM_DEVICE"   // DB37
{ S7_Optimized_Access := 'TRUE' }
VERSION : 0.1
// stored: AutoNumber true, DBAccessibleFromOPCUA true, DBAccessibleFromWebserver true, IsOnlyStoredInLoadMemory false, IsRetainMemResEnabled false, IsWriteProtectedInAS false, MemoryReserve 100
   VAR
      bannerStatus : Array[0..1023] of Bool;
      manifold : Array[0..1023] of Bool;
      iolink2 : Array[0..1023] of Bool;
      iolink1 : Array[0..1023] of Bool;
   END_VAR
BEGIN
   bannerStatus[0..1023] := FALSE;
   manifold[0..1023] := FALSE;
   iolink2[0] := TRUE;
   iolink2[1..5] := FALSE;
   iolink2[6] := TRUE;
   iolink2[7..1023] := FALSE;
   iolink1[0..1023] := FALSE;
END_DATA_BLOCK

ORGANIZATION_BLOCK "Main"   // OB1, LAD, ProgramCycle
TITLE = "Main Program Sweep (Cycle)"
{ S7_Optimized_Access := 'TRUE' }
VERSION : 0.1
// stored: AutoNumber true, IsIECCheckEnabled false, SetENOAutomatically false
   VAR_INPUT
      Initial_Call : Bool;   // Initial call of this OB
      Remanence : Bool;   // =True, if remanent data are available
   END_VAR
   VAR_TEMP
      BUFFER : String;
   END_VAR
   VAR_TEMP   // added for the SCL form of the ladder/FBD networks
      _w1 : Bool;
      _w2 : Bool;
      _w3 : Bool;
      _w4 : Bool;
      _w5 : Bool;
      _w6 : Bool;
      _w7 : Bool;
      _w8 : Bool;
      _w9 : Bool;
      _w10 : Bool;
      _w11 : Bool;
   END_VAR
BEGIN

REGION Network 1: SECUENCIA PARA ALARMAR LA MÁQUINA SI SE APAGA A LA MITAD DE UN CICLO DE PRODUCCIÓN
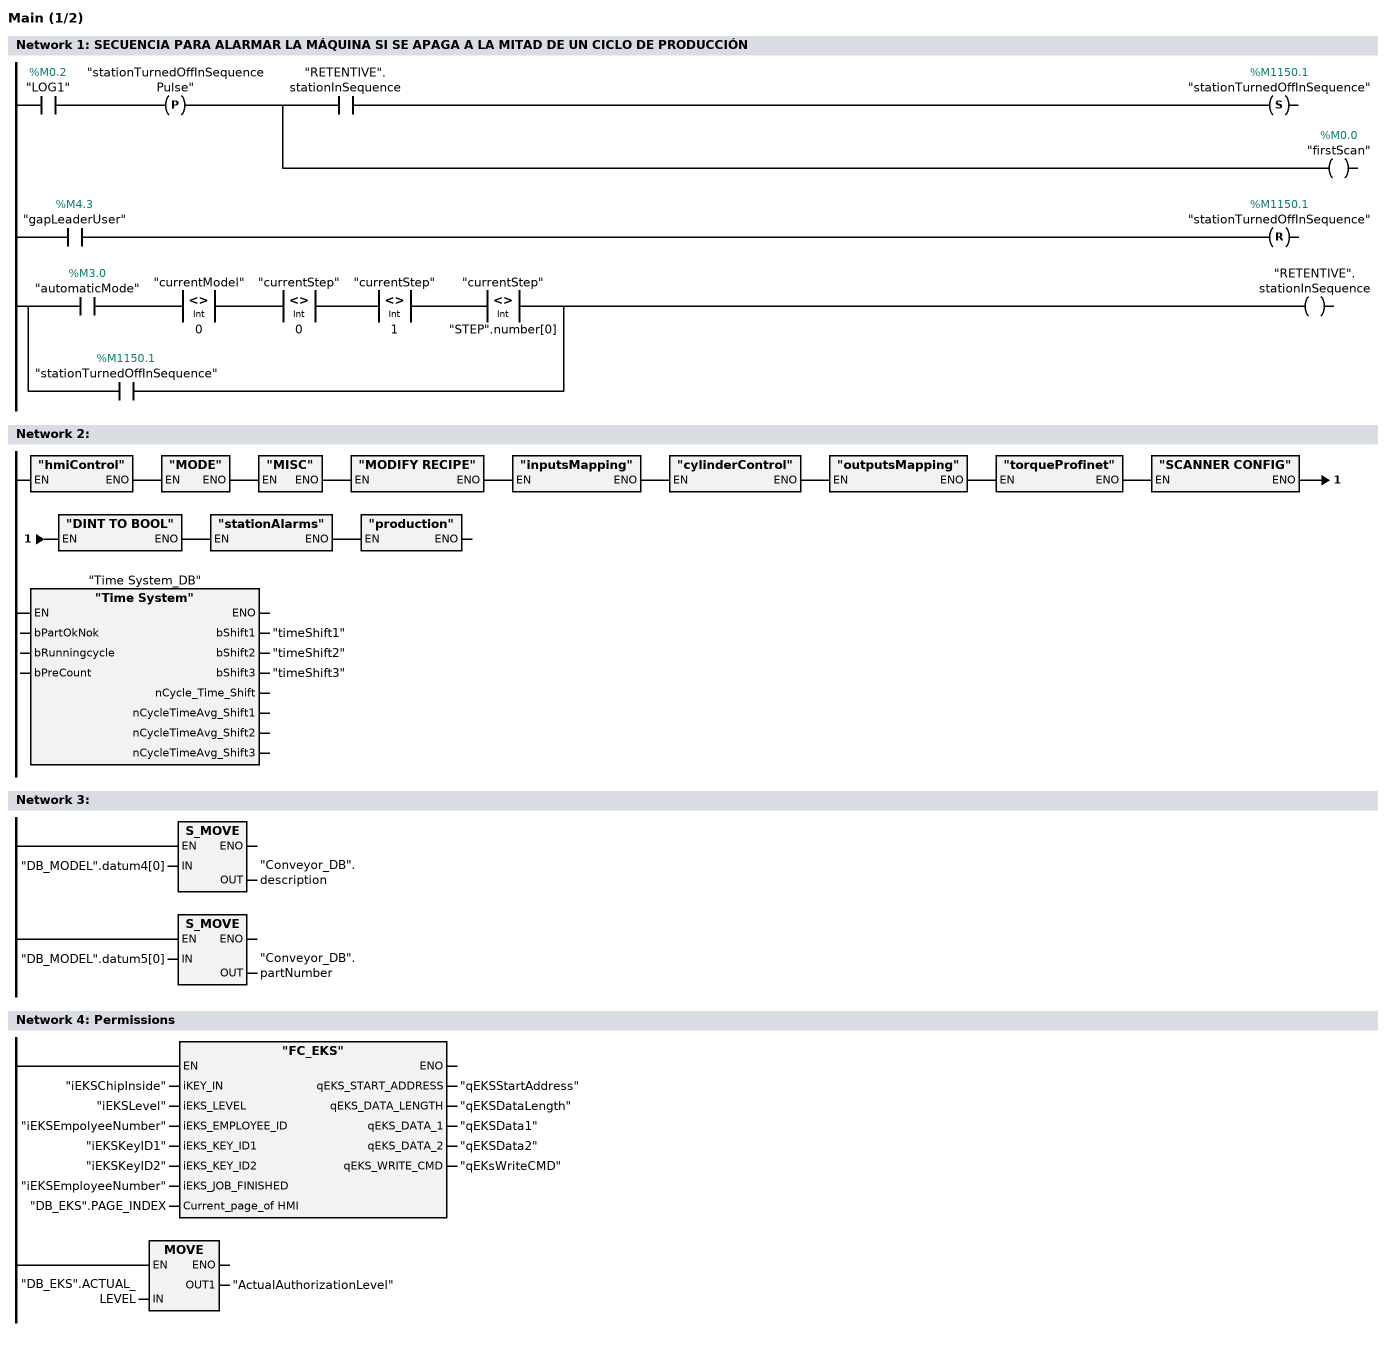
   RUNG wire#powerrail
      Contact( "LOG1" )
      P_Trig( "stationTurnedOffInSequencePulse" )
      wire#w1
      Contact( "RETENTIVE".stationInSequence )
      S_Coil( "stationTurnedOffInSequence" )
   END_RUNG
   RUNG wire#w1
      Coil( "firstScan" )
   END_RUNG
   RUNG wire#powerrail
      Contact( "gapLeaderUser" )
      R_Coil( "stationTurnedOffInSequence" )
   END_RUNG
   RUNG wire#powerrail
      Contact( "automaticMode" )
      { S7_Templates := "SrcType := Int" } NE_Contact(in1 := "currentModel", in2 := 0)
      { S7_Templates := "SrcType := Int" } NE_Contact(in1 := "currentStep", in2 := 0)
      { S7_Templates := "SrcType := Int" } NE_Contact(in1 := "currentStep", in2 := 1)
      { S7_Templates := "SrcType := Int" } NE_Contact(in1 := "currentStep", in2 := "STEP".number[0])
      wire#w2
      Coil( "RETENTIVE".stationInSequence )
   END_RUNG
   RUNG wire#powerrail
      Contact( "stationTurnedOffInSequence" )
   END_RUNG wire#w2
   // the same network as SCL:
   #_w1 := "LOG1" AND NOT "stationTurnedOffInSequencePulse";   // rising edge
   "stationTurnedOffInSequencePulse" := "LOG1";
   IF #_w1 AND "RETENTIVE".stationInSequence THEN "stationTurnedOffInSequence" := TRUE; END_IF;
   "firstScan" := #_w1;
   IF "gapLeaderUser" THEN "stationTurnedOffInSequence" := FALSE; END_IF;
   "RETENTIVE".stationInSequence := ("automaticMode" AND ("currentModel" <> 0) AND ("currentStep" <> 0) AND ("currentStep" <> 1) AND ("currentStep" <> "STEP".number[0])) OR "stationTurnedOffInSequence";
END_REGION

REGION Network 2
   RUNG wire#powerrail
      "hmiControl"()
      "MODE"()
      "MISC"()
      "MODIFY RECIPE"()
      "inputsMapping"()
      "cylinderControl"()
      "outputsMapping"()
      "torqueProfinet"()
      "SCANNER CONFIG"()
      "DINT TO BOOL"()
      "stationAlarms"()
      "production"()
   END_RUNG
   RUNG wire#powerrail
      "Time System_DB"(bPartOkNok :=, bRunningcycle :=, bPreCount :=, bShift1 => "timeShift1", bShift2 => "timeShift2", bShift3 => "timeShift3", nCycle_Time_Shift =>, nCycleTimeAvg_Shift1 =>, nCycleTimeAvg_Shift2 =>, nCycleTimeAvg_Shift3 =>)
   END_RUNG
   // the same network as SCL:
   "hmiControl"(ENO => #_w1);
   "MODE"(EN := #_w1, ENO => #_w2);
   "MISC"(EN := #_w2, ENO => #_w3);
   "MODIFY RECIPE"(EN := #_w3, ENO => #_w4);
   "inputsMapping"(EN := #_w4, ENO => #_w5);
   "cylinderControl"(EN := #_w5, ENO => #_w6);
   "outputsMapping"(EN := #_w6, ENO => #_w7);
   "torqueProfinet"(EN := #_w7, ENO => #_w8);
   "SCANNER CONFIG"(EN := #_w8, ENO => #_w9);
   "DINT TO BOOL"(EN := #_w9, ENO => #_w10);
   "stationAlarms"(EN := #_w10, ENO => #_w11);
   IF #_w11 THEN "production"(); END_IF;
   "Time System_DB"(bShift1 => "timeShift1", bShift2 => "timeShift2", bShift3 => "timeShift3");   // "Time System"
END_REGION

REGION Network 3
   RUNG wire#powerrail
      S_Move(in := "DB_MODEL".datum4[0], out => "Conveyor_DB".description)
   END_RUNG
   RUNG wire#powerrail
      S_Move(in := "DB_MODEL".datum5[0], out => "Conveyor_DB".partNumber)
   END_RUNG
   // the same network as SCL:
   "Conveyor_DB".description := "DB_MODEL".datum4[0];
   "Conveyor_DB".partNumber := "DB_MODEL".datum5[0];
END_REGION

REGION Network 4: Permissions
   RUNG wire#powerrail
      "FC_EKS"(iKEY_IN := "iEKSChipInside", iEKS_LEVEL := "iEKSLevel", iEKS_EMPLOYEE_ID := "iEKSEmpolyeeNumber", iEKS_KEY_ID1 := "iEKSKeyID1", iEKS_KEY_ID2 := "iEKSKeyID2", iEKS_JOB_FINISHED := "iEKSEmployeeNumber", "Current_page_of HMI" := "DB_EKS".PAGE_INDEX, qEKS_START_ADDRESS => "qEKSStartAddress", qEKS_DATA_LENGTH => "qEKSDataLength", qEKS_DATA_1 => "qEKSData1", qEKS_DATA_2 => "qEKSData2", qEKS_WRITE_CMD => "qEKsWriteCMD")
   END_RUNG
   RUNG wire#powerrail
      Move(in := "DB_EKS".ACTUAL_LEVEL, out1 => "ActualAuthorizationLevel")
   END_RUNG
   // the same network as SCL:
   "FC_EKS"(iKEY_IN := "iEKSChipInside",
            iEKS_LEVEL := "iEKSLevel",
            iEKS_EMPLOYEE_ID := "iEKSEmpolyeeNumber",
            iEKS_KEY_ID1 := "iEKSKeyID1",
            iEKS_KEY_ID2 := "iEKSKeyID2",
            iEKS_JOB_FINISHED := "iEKSEmployeeNumber",
            "Current_page_of HMI" := "DB_EKS".PAGE_INDEX,
            qEKS_START_ADDRESS => "qEKSStartAddress",
            qEKS_DATA_LENGTH => "qEKSDataLength",
            qEKS_DATA_1 => "qEKSData1",
            qEKS_DATA_2 => "qEKSData2",
            qEKS_WRITE_CMD => "qEKsWriteCMD");
   "ActualAuthorizationLevel" := "DB_EKS".ACTUAL_LEVEL;
END_REGION

REGION Network 5: Awake signal
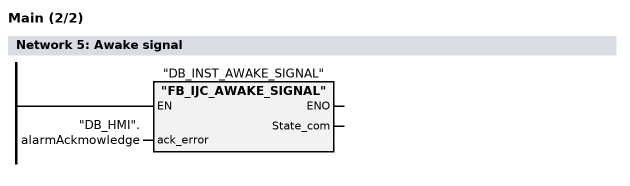
   RUNG wire#powerrail
      "DB_INST_AWAKE_SIGNAL"(ack_error := "DB_HMI".alarmAckmowledge, State_com =>)
   END_RUNG
   // the same network as SCL:
   "DB_INST_AWAKE_SIGNAL"(ack_error := "DB_HMI".alarmAckmowledge);   // "FB_IJC_AWAKE_SIGNAL"
END_REGION
END_ORGANIZATION_BLOCK

FUNCTION "hmiControl" : Void   // FC3, LAD
{ S7_Optimized_Access := 'TRUE' }
VERSION : 0.1
// stored: AutoNumber true, IsIECCheckEnabled false, SetENOAutomatically false, UDAEnableTagReadback false
   VAR_TEMP   // added for the SCL form of the ladder/FBD networks
      _w1 : Bool;
      _w2 : Bool;
      _w3 : Bool;
      _w4 : Bool;
      _w5 : Bool;
      _w6 : Bool;
      _w7 : Bool;
      _w8 : Bool;
      _w9 : Bool;
      _w10 : Bool;
      _w11 : Bool;
      _w12 : Bool;
      _w13 : Bool;
      _w14 : Bool;
      _w15 : Bool;
      _w16 : Bool;
      _w17 : Bool;
      _w18 : Bool;
      _w19 : Bool;
      _w20 : Bool;
      _w21 : Bool;
      _w22 : Bool;
      _w23 : Bool;
      _w24 : Bool;
      _w25 : Bool;
      _w26 : Bool;
      _w27 : Bool;
      _w28 : Bool;
      _w29 : Bool;
      _w30 : Bool;
      _w31 : Bool;
      _w32 : Bool;
   END_VAR
BEGIN

REGION Network 1: VISUALIZACIÓN DE MODELOS: SI CADA MODELO TIENE UN NOMBRE GRABADO, SE ACTIVA SU VISUALIZACIÓN
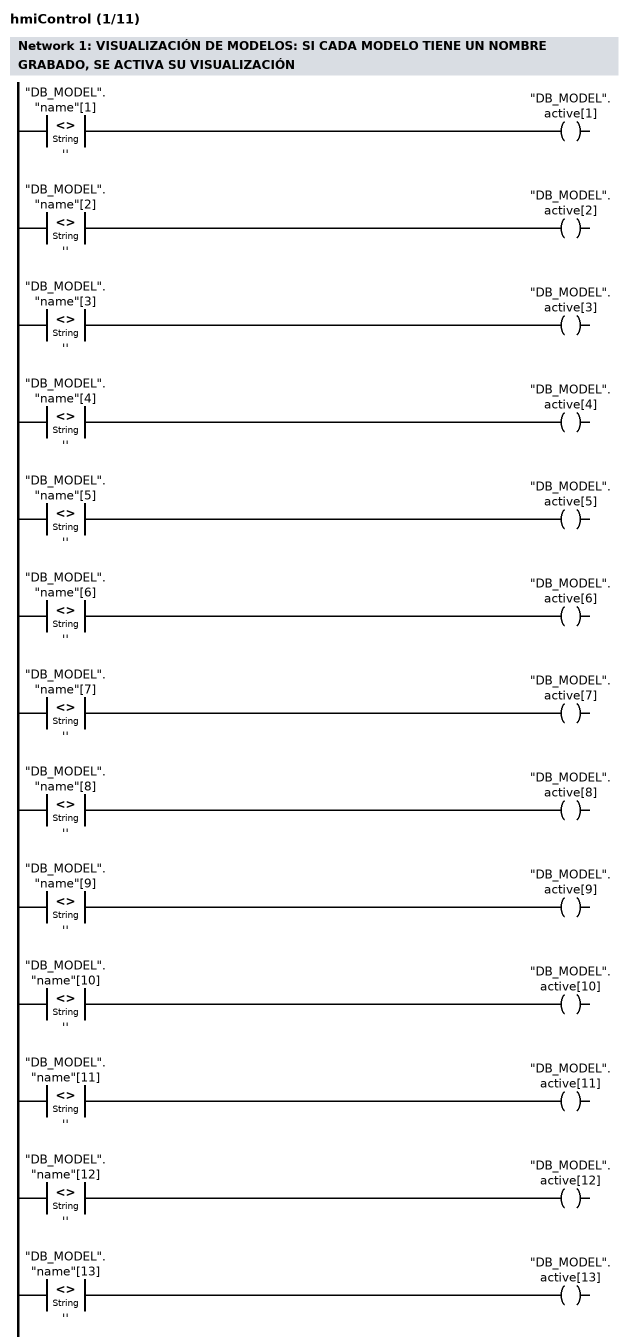
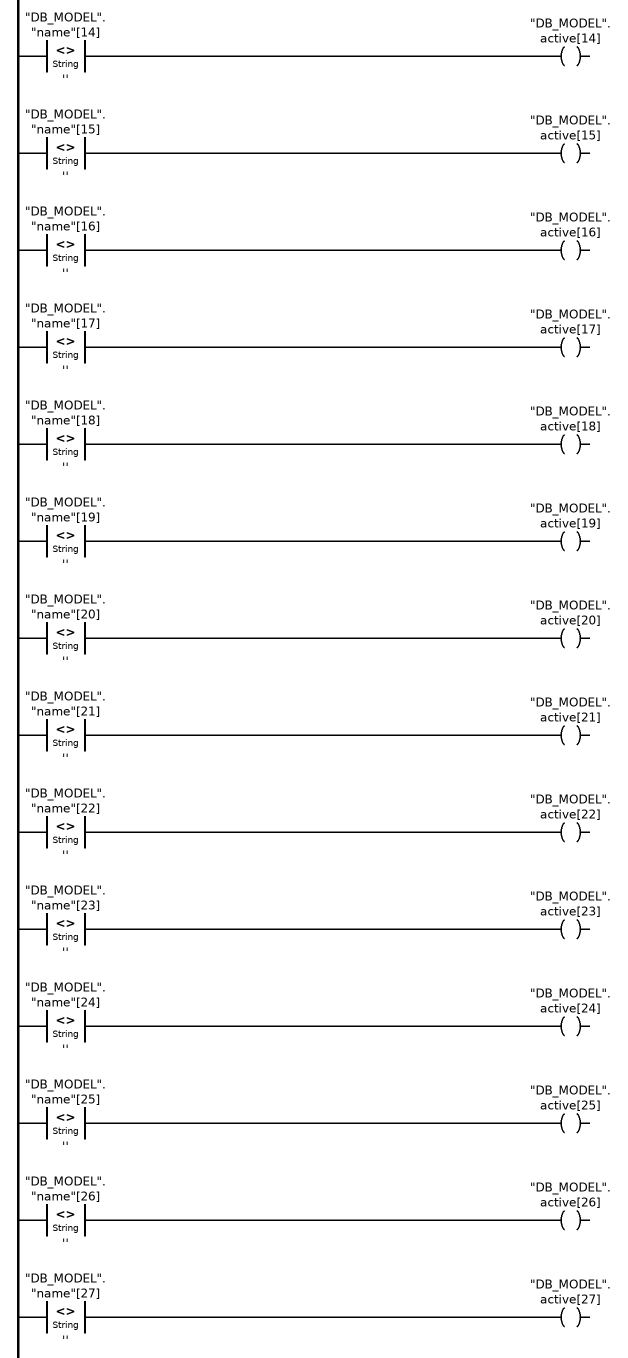
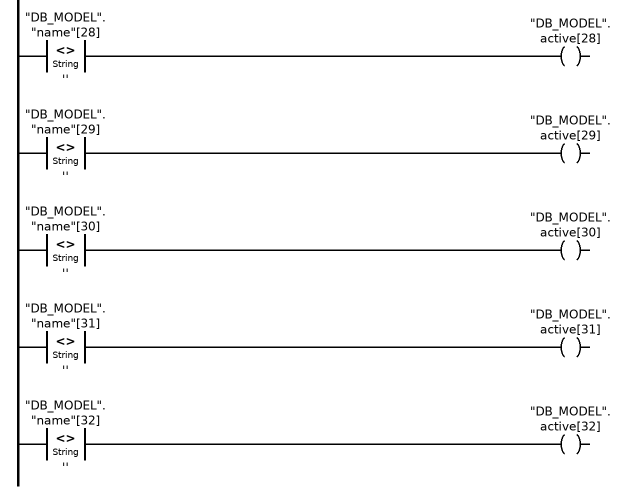
   RUNG wire#powerrail
      { S7_Templates := "SrcType := String" } NE_Contact(in1 := "DB_MODEL"."name"[1], in2 := '')
      Coil( "DB_MODEL".active[1] )
   END_RUNG
   RUNG wire#powerrail
      { S7_Templates := "SrcType := String" } NE_Contact(in1 := "DB_MODEL"."name"[2], in2 := '')
      Coil( "DB_MODEL".active[2] )
   END_RUNG
   RUNG wire#powerrail
      { S7_Templates := "SrcType := String" } NE_Contact(in1 := "DB_MODEL"."name"[3], in2 := '')
      Coil( "DB_MODEL".active[3] )
   END_RUNG
   RUNG wire#powerrail
      { S7_Templates := "SrcType := String" } NE_Contact(in1 := "DB_MODEL"."name"[4], in2 := '')
      Coil( "DB_MODEL".active[4] )
   END_RUNG
   RUNG wire#powerrail
      { S7_Templates := "SrcType := String" } NE_Contact(in1 := "DB_MODEL"."name"[5], in2 := '')
      Coil( "DB_MODEL".active[5] )
   END_RUNG
   RUNG wire#powerrail
      { S7_Templates := "SrcType := String" } NE_Contact(in1 := "DB_MODEL"."name"[6], in2 := '')
      Coil( "DB_MODEL".active[6] )
   END_RUNG
   RUNG wire#powerrail
      { S7_Templates := "SrcType := String" } NE_Contact(in1 := "DB_MODEL"."name"[7], in2 := '')
      Coil( "DB_MODEL".active[7] )
   END_RUNG
   RUNG wire#powerrail
      { S7_Templates := "SrcType := String" } NE_Contact(in1 := "DB_MODEL"."name"[8], in2 := '')
      Coil( "DB_MODEL".active[8] )
   END_RUNG
   RUNG wire#powerrail
      { S7_Templates := "SrcType := String" } NE_Contact(in1 := "DB_MODEL"."name"[9], in2 := '')
      Coil( "DB_MODEL".active[9] )
   END_RUNG
   RUNG wire#powerrail
      { S7_Templates := "SrcType := String" } NE_Contact(in1 := "DB_MODEL"."name"[10], in2 := '')
      Coil( "DB_MODEL".active[10] )
   END_RUNG
   RUNG wire#powerrail
      { S7_Templates := "SrcType := String" } NE_Contact(in1 := "DB_MODEL"."name"[11], in2 := '')
      Coil( "DB_MODEL".active[11] )
   END_RUNG
   RUNG wire#powerrail
      { S7_Templates := "SrcType := String" } NE_Contact(in1 := "DB_MODEL"."name"[12], in2 := '')
      Coil( "DB_MODEL".active[12] )
   END_RUNG
   RUNG wire#powerrail
      { S7_Templates := "SrcType := String" } NE_Contact(in1 := "DB_MODEL"."name"[13], in2 := '')
      Coil( "DB_MODEL".active[13] )
   END_RUNG
   RUNG wire#powerrail
      { S7_Templates := "SrcType := String" } NE_Contact(in1 := "DB_MODEL"."name"[14], in2 := '')
      Coil( "DB_MODEL".active[14] )
   END_RUNG
   RUNG wire#powerrail
      { S7_Templates := "SrcType := String" } NE_Contact(in1 := "DB_MODEL"."name"[15], in2 := '')
      Coil( "DB_MODEL".active[15] )
   END_RUNG
   RUNG wire#powerrail
      { S7_Templates := "SrcType := String" } NE_Contact(in1 := "DB_MODEL"."name"[16], in2 := '')
      Coil( "DB_MODEL".active[16] )
   END_RUNG
   RUNG wire#powerrail
      { S7_Templates := "SrcType := String" } NE_Contact(in1 := "DB_MODEL"."name"[17], in2 := '')
      Coil( "DB_MODEL".active[17] )
   END_RUNG
   RUNG wire#powerrail
      { S7_Templates := "SrcType := String" } NE_Contact(in1 := "DB_MODEL"."name"[18], in2 := '')
      Coil( "DB_MODEL".active[18] )
   END_RUNG
   RUNG wire#powerrail
      { S7_Templates := "SrcType := String" } NE_Contact(in1 := "DB_MODEL"."name"[19], in2 := '')
      Coil( "DB_MODEL".active[19] )
   END_RUNG
   RUNG wire#powerrail
      { S7_Templates := "SrcType := String" } NE_Contact(in1 := "DB_MODEL"."name"[20], in2 := '')
      Coil( "DB_MODEL".active[20] )
   END_RUNG
   RUNG wire#powerrail
      { S7_Templates := "SrcType := String" } NE_Contact(in1 := "DB_MODEL"."name"[21], in2 := '')
      Coil( "DB_MODEL".active[21] )
   END_RUNG
   RUNG wire#powerrail
      { S7_Templates := "SrcType := String" } NE_Contact(in1 := "DB_MODEL"."name"[22], in2 := '')
      Coil( "DB_MODEL".active[22] )
   END_RUNG
   RUNG wire#powerrail
      { S7_Templates := "SrcType := String" } NE_Contact(in1 := "DB_MODEL"."name"[23], in2 := '')
      Coil( "DB_MODEL".active[23] )
   END_RUNG
   RUNG wire#powerrail
      { S7_Templates := "SrcType := String" } NE_Contact(in1 := "DB_MODEL"."name"[24], in2 := '')
      Coil( "DB_MODEL".active[24] )
   END_RUNG
   RUNG wire#powerrail
      { S7_Templates := "SrcType := String" } NE_Contact(in1 := "DB_MODEL"."name"[25], in2 := '')
      Coil( "DB_MODEL".active[25] )
   END_RUNG
   RUNG wire#powerrail
      { S7_Templates := "SrcType := String" } NE_Contact(in1 := "DB_MODEL"."name"[26], in2 := '')
      Coil( "DB_MODEL".active[26] )
   END_RUNG
   RUNG wire#powerrail
      { S7_Templates := "SrcType := String" } NE_Contact(in1 := "DB_MODEL"."name"[27], in2 := '')
      Coil( "DB_MODEL".active[27] )
   END_RUNG
   RUNG wire#powerrail
      { S7_Templates := "SrcType := String" } NE_Contact(in1 := "DB_MODEL"."name"[28], in2 := '')
      Coil( "DB_MODEL".active[28] )
   END_RUNG
   RUNG wire#powerrail
      { S7_Templates := "SrcType := String" } NE_Contact(in1 := "DB_MODEL"."name"[29], in2 := '')
      Coil( "DB_MODEL".active[29] )
   END_RUNG
   RUNG wire#powerrail
      { S7_Templates := "SrcType := String" } NE_Contact(in1 := "DB_MODEL"."name"[30], in2 := '')
      Coil( "DB_MODEL".active[30] )
   END_RUNG
   RUNG wire#powerrail
      { S7_Templates := "SrcType := String" } NE_Contact(in1 := "DB_MODEL"."name"[31], in2 := '')
      Coil( "DB_MODEL".active[31] )
   END_RUNG
   RUNG wire#powerrail
      { S7_Templates := "SrcType := String" } NE_Contact(in1 := "DB_MODEL"."name"[32], in2 := '')
      Coil( "DB_MODEL".active[32] )
   END_RUNG
   // the same network as SCL:
   "DB_MODEL".active[1] := "DB_MODEL"."name"[1] <> '';
   "DB_MODEL".active[2] := "DB_MODEL"."name"[2] <> '';
   "DB_MODEL".active[3] := "DB_MODEL"."name"[3] <> '';
   "DB_MODEL".active[4] := "DB_MODEL"."name"[4] <> '';
   "DB_MODEL".active[5] := "DB_MODEL"."name"[5] <> '';
   "DB_MODEL".active[6] := "DB_MODEL"."name"[6] <> '';
   "DB_MODEL".active[7] := "DB_MODEL"."name"[7] <> '';
   "DB_MODEL".active[8] := "DB_MODEL"."name"[8] <> '';
   "DB_MODEL".active[9] := "DB_MODEL"."name"[9] <> '';
   "DB_MODEL".active[10] := "DB_MODEL"."name"[10] <> '';
   "DB_MODEL".active[11] := "DB_MODEL"."name"[11] <> '';
   "DB_MODEL".active[12] := "DB_MODEL"."name"[12] <> '';
   "DB_MODEL".active[13] := "DB_MODEL"."name"[13] <> '';
   "DB_MODEL".active[14] := "DB_MODEL"."name"[14] <> '';
   "DB_MODEL".active[15] := "DB_MODEL"."name"[15] <> '';
   "DB_MODEL".active[16] := "DB_MODEL"."name"[16] <> '';
   "DB_MODEL".active[17] := "DB_MODEL"."name"[17] <> '';
   "DB_MODEL".active[18] := "DB_MODEL"."name"[18] <> '';
   "DB_MODEL".active[19] := "DB_MODEL"."name"[19] <> '';
   "DB_MODEL".active[20] := "DB_MODEL"."name"[20] <> '';
   "DB_MODEL".active[21] := "DB_MODEL"."name"[21] <> '';
   "DB_MODEL".active[22] := "DB_MODEL"."name"[22] <> '';
   "DB_MODEL".active[23] := "DB_MODEL"."name"[23] <> '';
   "DB_MODEL".active[24] := "DB_MODEL"."name"[24] <> '';
   "DB_MODEL".active[25] := "DB_MODEL"."name"[25] <> '';
   "DB_MODEL".active[26] := "DB_MODEL"."name"[26] <> '';
   "DB_MODEL".active[27] := "DB_MODEL"."name"[27] <> '';
   "DB_MODEL".active[28] := "DB_MODEL"."name"[28] <> '';
   "DB_MODEL".active[29] := "DB_MODEL"."name"[29] <> '';
   "DB_MODEL".active[30] := "DB_MODEL"."name"[30] <> '';
   "DB_MODEL".active[31] := "DB_MODEL"."name"[31] <> '';
   "DB_MODEL".active[32] := "DB_MODEL"."name"[32] <> '';
END_REGION

REGION Network 2: CURRENT MODEL NAME SHOWN IN HMI
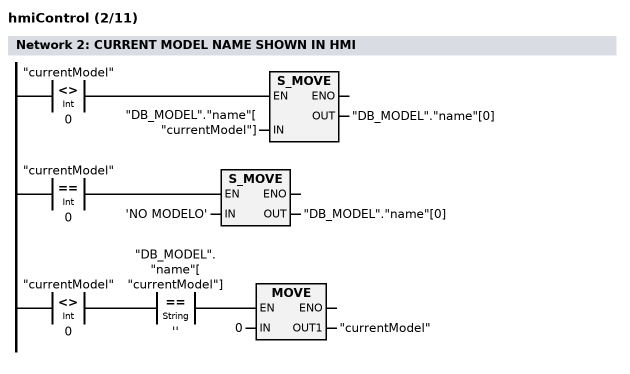
   RUNG wire#powerrail
      { S7_Templates := "SrcType := Int" } NE_Contact(in1 := "currentModel", in2 := 0)
      S_Move(in := "DB_MODEL"."name"["currentModel"], out => "DB_MODEL"."name"[0])
   END_RUNG
   RUNG wire#powerrail
      { S7_Templates := "SrcType := Int" } EQ_Contact(in1 := "currentModel", in2 := 0)
      S_Move(in := 'NO MODELO', out => "DB_MODEL"."name"[0])
   END_RUNG
   RUNG wire#powerrail
      { S7_Templates := "SrcType := Int" } NE_Contact(in1 := "currentModel", in2 := 0)
      { S7_Templates := "SrcType := String" } EQ_Contact(in1 := "DB_MODEL"."name"["currentModel"], in2 := '')
      Move(in := 0, out1 => "currentModel")
   END_RUNG
   // the same network as SCL:
   IF "currentModel" <> 0 THEN "DB_MODEL"."name"[0] := "DB_MODEL"."name"["currentModel"]; END_IF;
   IF "currentModel" = 0 THEN "DB_MODEL"."name"[0] := 'NO MODELO'; END_IF;
   IF ("currentModel" <> 0) AND ("DB_MODEL"."name"["currentModel"] = '') THEN "currentModel" := 0; END_IF;
END_REGION

